LIN {X 0,Y 362.905,Z 706.892,A -85,B 0,C 180,E1 -22587.78,E2 -22587.78} C_VEL
LIN {X 0,Y 363.363,Z 707.01,A -85,B 0,C 180,E1 -22590,E2 -22590} C_VEL
LIN {X 0,Y 362.89,Z 706.909,A -85,B 0,C 180,E1 -22592.22,E2 -22592.22} C_VEL
LIN {X 0,Y 362.378,Z 706.638,A -85,B 0,C 180,E1 -22593.335,E2 -22593.335} C_VEL
LIN {X 0,Y 360.579,Z 706.015,A -85,B 0,C 180,E1 -22595.592,E2 -22595.592} C_VEL
LIN {X 0,Y 357.963,Z 704.809,A -85,B 0,C 180,E1 -22597.899,E2 -22597.899} C_VEL
LIN {X 0,Y 356.048,Z 703.774,A -85,B 0,C 180,E1 -22599.273,E2 -22599.273} C_VEL
LIN {X 0,Y 352.322,Z 701.531,A -85,B 0,C 180,E1 -22601.506,E2 -22601.506} C_VEL
LIN {X 0,Y 349.963,Z 699.883,A -85,B 0,C 180,E1 -22602.762,E2 -22602.762} C_VEL
LIN {X 0,Y 347.344,Z 697.848,A -85,B 0,C 180,E1 -22604.052,E2 -22604.052} C_VEL
LIN {X 0,Y 343.234,Z 695.3,A -85,B 0,C 180,E1 -22605.772,E2 -22605.772} C_VEL
LIN {X 0,Y 338.777,Z 692.643,A -85,B 0,C 180,E1 -22607.395,E2 -22607.395} C_VEL
LIN {X 0,Y 332.769,Z 688.318,A -85,B 0,C 180,E1 -22609.499,E2 -22609.499} C_VEL
LIN {X 0,Y 328.202,Z 685.08,A -85,B 0,C 180,E1 -22610.918,E2 -22610.918} C_VEL
LIN {X 0,Y 320.695,Z 679.914,A -85,B 0,C 180,E1 -22613.014,E2 -22613.014} C_VEL
LIN {X 0,Y 313.527,Z 674.664,A -85,B 0,C 180,E1 -22614.877,E2 -22614.877} C_VEL
LIN {X 0,Y 306.386,Z 669.423,A -85,B 0,C 180,E1 -22616.545,E2 -22616.545} C_VEL
LIN {X 0,Y 300.005,Z 664.622,A -85,B 0,C 180,E1 -22617.938,E2 -22617.938} C_VEL
LIN {X 0,Y 291.37,Z 657.885,A -85,B 0,C 180,E1 -22619.648,E2 -22619.648} C_VEL
LIN {X 0,Y 281.833,Z 650.578,A -85,B 0,C 180,E1 -22621.3,E2 -22621.3} C_VEL
LIN {X 0,Y 269.07,Z 639.844,A -85,B 0,C 180,E1 -22623.529,E2 -22623.529} C_VEL
LIN {X 0,Y 258.955,Z 630.539,A -85,B 0,C 180,E1 -22625.379,E2 -22625.379} C_VEL
LIN {X 0,Y 245.067,Z 616.202,A -85,B 0,C 180,E1 -22628.261,E2 -22628.261} C_VEL
LIN {X 0,Y 234.328,Z 603.001,A -85,B 0,C 180,E1 -22630.902,E2 -22630.902} C_VEL
LIN {X 0,Y 225.204,Z 588.908,A -85,B 0,C 180,E1 -22633.566,E2 -22633.566} C_VEL
LIN {X 0,Y 214.798,Z 569.008,A -85,B 0,C 180,E1 -22637.242,E2 -22637.242} C_VEL
LIN {X 0,Y 207.799,Z 557.073,A -85,B 0,C 180,E1 -22640.015,E2 -22640.015} C_VEL
LIN {X 0,Y 200.862,Z 546.571,A -85,B 0,C 180,E1 -22643.065,E2 -22643.065} C_VEL
LIN {X 0,Y 196.487,Z 540.686,A -85,B 0,C 180,E1 -22645.179,E2 -22645.179} C_VEL
LIN {X 0,Y 194.374,Z 537.758,A -85,B 0,C 180,E1 -22646.283,E2 -22646.283} C_VEL
LIN {X 0,Y 191.516,Z 533.827,A -85,B 0,C 180,E1 -22647.868,E2 -22647.868} C_VEL
LIN {X 0,Y 188.498,Z 530.398,A -85,B 0,C 180,E1 -22649.626,E2 -22649.626} C_VEL
LIN {X 0,Y 187.385,Z 528.546,A -85,B 0,C 180,E1 -22650.357,E2 -22650.357} C_VEL
LIN {X 0,Y 184.854,Z 526.226,A -85,B 0,C 180,E1 -22651.967,E2 -22651.967} C_VEL
LIN {X 0,Y 183.022,Z 523.18,A -85,B 0,C 180,E1 -22653.335,E2 -22653.335} C_VEL
LIN {X 0,Y 180.33,Z 521.243,A -85,B 0,C 180,E1 -22655.289,E2 -22655.289} C_VEL
LIN {X 0,Y 178.835,Z 518.728,A -85,B 0,C 180,E1 -22656.65,E2 -22656.65} C_VEL
LIN {X 0,Y 178.593,Z 517.589,A -85,B 0,C 180,E1 -22657.516,E2 -22657.516} C_VEL
LIN {X 0,Y 178.645,Z 517.32,A -85,B 0,C 180,E1 -22661.657,E2 -22661.657} C_VEL
LIN {X 0,Y 178.652,Z 517.357,A -85,B 0,C 180,E1 -22666.349,E2 -22666.349} C_VEL
LIN {X 0,Y 178.907,Z 517.281,A -85,B 0,C 180,E1 -22670.961,E2 -22670.961} C_VEL
LIN {X 0,Y 178.862,Z 517.301,A -85,B 0,C 180,E1 -22675.494,E2 -22675.494} C_VEL
LIN {X 0,Y 179.366,Z 517.233,A -85,B 0,C 180,E1 -22680.001,E2 -22680.001} C_VEL
LIN {X 0,Y 178.866,Z 517.288,A -85,B 0,C 180,E1 -22684.508,E2 -22684.508} C_VEL
LIN {X 0,Y 178.956,Z 517.309,A -85,B 0,C 180,E1 -22689.039,E2 -22689.039} C_VEL
LIN {X 0,Y 178.657,Z 517.313,A -85,B 0,C 180,E1 -22693.653,E2 -22693.653} C_VEL
LIN {X 0,Y 178.619,Z 517.329,A -85,B 0,C 180,E1 -22699.215,E2 -22699.215} C_VEL
LIN {X 0,Y 178.603,Z 517.694,A -85,B 0,C 180,E1 -22702.257,E2 -22702.257} C_VEL
LIN {X 0,Y 178.855,Z 518.824,A -85,B 0,C 180,E1 -22702.986,E2 -22702.986} C_VEL
LIN {X 0,Y 180.307,Z 521.22,A -85,B 0,C 180,E1 -22704.3,E2 -22704.3} C_VEL
LIN {X 0,Y 182.575,Z 522.942,A -85,B 0,C 180,E1 -22705.969,E2 -22705.969} C_VEL
LIN {X 0,Y 183.29,Z 523.542,A -85,B 0,C 180,E1 -22706.472,E2 -22706.472} C_VEL
LIN {X 0,Y 185.238,Z 526.708,A -85,B 0,C 180,E1 -22707.904,E2 -22707.904} C_VEL
LIN {X 0,Y 187.677,Z 528.97,A -85,B 0,C 180,E1 -22709.44,E2 -22709.44} C_VEL
LIN {X 0,Y 190.188,Z 532.55,A -85,B 0,C 180,E1 -22711.001,E2 -22711.001} C_VEL
LIN {X 0,Y 191.704,Z 534.216,A -85,B 0,C 180,E1 -22711.856,E2 -22711.856} C_VEL
LIN {X 0,Y 194.572,Z 537.949,A -85,B 0,C 180,E1 -22713.425,E2 -22713.425} C_VEL
LIN {X 0,Y 198.501,Z 544.029,A -85,B 0,C 180,E1 -22715.465,E2 -22715.465} C_VEL
LIN {X 0,Y 203.758,Z 553.106,A -85,B 0,C 180,E1 -22717.987,E2 -22717.987} C_VEL
LIN {X 0,Y 209.85,Z 564.904,A -85,B 0,C 180,E1 -22720.663,E2 -22720.663} C_VEL
LIN {X 0,Y 215.674,Z 577.872,A -85,B 0,C 180,E1 -22723.042,E2 -22723.042} C_VEL
LIN {X 0,Y 220.269,Z 589.701,A -85,B 0,C 180,E1 -22724.835,E2 -22724.835} C_VEL
LIN {X 0,Y 216.464,Z 650.604,A -85,B 0,C 180,E1 -22726.656,E2 -22726.656} C_VEL
LIN {X 0,Y 215.159,Z 662.058,A -85,B 0,C 180,E1 -22727.171,E2 -22727.171} C_VEL
LIN {X 0,Y 213.613,Z 671.685,A -85,B 0,C 180,E1 -22727.748,E2 -22727.748} C_VEL
LIN {X 0,Y 211.279,Z 682.832,A -85,B 0,C 180,E1 -22728.616,E2 -22728.616} C_VEL
LIN {X 0,Y 208.839,Z 692.8,A -85,B 0,C 180,E1 -22729.624,E2 -22729.624} C_VEL
LIN {X 0,Y 206.009,Z 702.716,A -85,B 0,C 180,E1 -22730.868,E2 -22730.868} C_VEL
LIN {X 0,Y 202.81,Z 712.435,A -85,B 0,C 180,E1 -22732.356,E2 -22732.356} C_VEL
LIN {X 0,Y 199.59,Z 721.567,A -85,B 0,C 180,E1 -22734.086,E2 -22734.086} C_VEL
LIN {X 0,Y 195.973,Z 730.873,A -85,B 0,C 180,E1 -22736.231,E2 -22736.231} C_VEL
LIN {X 0,Y 192.94,Z 737.844,A -85,B 0,C 180,E1 -22738.119,E2 -22738.119} C_VEL
LIN {X 0,Y 189.528,Z 745.364,A -85,B 0,C 180,E1 -22740.573,E2 -22740.573} C_VEL
LIN {X 0,Y 185.961,Z 752.975,A -85,B 0,C 180,E1 -22743.637,E2 -22743.637} C_VEL
LIN {X 0,Y 183.399,Z 758.378,A -85,B 0,C 180,E1 -22746.274,E2 -22746.274} C_VEL
LIN {X 0,Y 180.937,Z 763.817,A -85,B 0,C 180,E1 -22749.539,E2 -22749.539} C_VEL
LIN {X 0,Y 178.939,Z 768.266,A -85,B 0,C 180,E1 -22752.869,E2 -22752.869} C_VEL
LIN {X 0,Y 178.633,Z 768.942,A -85,B 0,C 180,E1 -22753.466,E2 -22753.466} C_VEL
LIN {X 0,Y 177.192,Z 770.925,A -85,B 0,C 180,E1 -22755.207,E2 -22755.207} C_VEL
LIN {X 0,Y 173.38,Z 773.511,A -85,B 0,C 180,E1 -22758.07,E2 -22758.07} C_VEL
LIN {X 0,Y 170.438,Z 775.159,A -85,B 0,C 180,E1 -22760.475,E2 -22760.475} C_VEL
LIN {X 0,Y 169.124,Z 776.109,A -85,B 0,C 180,E1 -22762.401,E2 -22762.401} C_VEL
LIN {X 0,Y 168.971,Z 776.341,A -85,B 0,C 180,E1 -22763.064,E2 -22763.064} C_VEL
LIN {X 0,Y 168.89,Z 777.565,A -85,B 0,C 180,E1 -22767.615,E2 -22767.615} C_VEL
LIN {X 0,Y 168.989,Z 777.822,A -85,B 0,C 180,E1 -22770,E2 -22770} C_VEL
LIN {X 0,Y 168.876,Z 777.085,A -85,B 0,C 180,E1 -22774.774,E2 -22774.774} C_VEL
LIN {X 0,Y 168.995,Z 776.261,A -85,B 0,C 180,E1 -22777.167,E2 -22777.167} C_VEL
LIN {X 0,Y 169.781,Z 773.563,A -85,B 0,C 180,E1 -22781.945,E2 -22781.945} C_VEL
LIN {X 0,Y 171.508,Z 769.334,A -85,B 0,C 180,E1 -22786.669,E2 -22786.669} C_VEL
LIN {X 0,Y 173.456,Z 765.197,A -85,B 0,C 180,E1 -22790.145,E2 -22790.145} C_VEL
LIN {X 0,Y 175.898,Z 760.093,A -85,B 0,C 180,E1 -22793.549,E2 -22793.549} C_VEL
LIN {X 0,Y 178.995,Z 753.913,A -85,B 0,C 180,E1 -22796.841,E2 -22796.841} C_VEL
LIN {X 0,Y 182.03,Z 747.84,A -85,B 0,C 180,E1 -22799.489,E2 -22799.489} C_VEL
LIN {X 0,Y 185.435,Z 740.767,A -85,B 0,C 180,E1 -22802.045,E2 -22802.045} C_VEL
LIN {X 0,Y 188.506,Z 734.31,A -85,B 0,C 180,E1 -22804.002,E2 -22804.002} C_VEL
LIN {X 0,Y 192.369,Z 725.334,A -85,B 0,C 180,E1 -22806.264,E2 -22806.264} C_VEL
LIN {X 0,Y 195.922,Z 715.957,A -85,B 0,C 180,E1 -22808.226,E2 -22808.226} C_VEL
LIN {X 0,Y 199.134,Z 706.91,A -85,B 0,C 180,E1 -22809.767,E2 -22809.767} C_VEL
LIN {X 0,Y 202.473,Z 696.107,A -85,B 0,C 180,E1 -22811.261,E2 -22811.261} C_VEL
LIN {X 0,Y 205.254,Z 685.854,A -85,B 0,C 180,E1 -22812.384,E2 -22812.384} C_VEL
LIN {X 0,Y 207.849,Z 674.205,A -85,B 0,C 180,E1 -22813.378,E2 -22813.378} C_VEL
LIN {X 0,Y 209.834,Z 662.77,A -85,B 0,C 180,E1 -22814.108,E2 -22814.108} C_VEL
LIN {X 0,Y 211.198,Z 651.913,A -85,B 0,C 180,E1 -22814.603,E2 -22814.603} C_VEL
LIN {X 0,Y 212.886,Z 628.702,A -85,B 0,C 180,E1 -22815.328,E2 -22815.328} C_VEL
LIN {X 0,Y 215.147,Z 591.855,A -85,B 0,C 180,E1 -22816.442,E2 -22816.442} C_VEL
LIN {X 0,Y 210.265,Z 579.231,A -85,B 0,C 180,E1 -22818.481,E2 -22818.481} C_VEL
LIN {X 0,Y 204.814,Z 567.17,A -85,B 0,C 180,E1 -22820.871,E2 -22820.871} C_VEL
LIN {X 0,Y 199.071,Z 556.016,A -85,B 0,C 180,E1 -22823.59,E2 -22823.59} C_VEL
LIN {X 0,Y 193.918,Z 547.035,A -85,B 0,C 180,E1 -22826.272,E2 -22826.272} C_VEL
LIN {X 0,Y 191.631,Z 543.666,A -85,B 0,C 180,E1 -22827.531,E2 -22827.531} C_VEL
LIN {X 0,Y 188.143,Z 539.098,A -85,B 0,C 180,E1 -22829.56,E2 -22829.56} C_VEL
LIN {X 0,Y 185.338,Z 535.278,A -85,B 0,C 180,E1 -22831.356,E2 -22831.356} C_VEL
LIN {X 0,Y 182.1,Z 531.683,A -85,B 0,C 180,E1 -22833.573,E2 -22833.573} C_VEL
LIN {X 0,Y 180.96,Z 529.723,A -85,B 0,C 180,E1 -22834.477,E2 -22834.477} C_VEL
LIN {X 0,Y 178.143,Z 527.388,A -85,B 0,C 180,E1 -22836.658,E2 -22836.658} C_VEL
LIN {X 0,Y 176.353,Z 524.222,A -85,B 0,C 180,E1 -22838.368,E2 -22838.368} C_VEL
LIN {X 0,Y 173.51,Z 522.23,A -85,B 0,C 180,E1 -22841.092,E2 -22841.092} C_VEL
LIN {X 0,Y 171.922,Z 519.752,A -85,B 0,C 180,E1 -22843.065,E2 -22843.065} C_VEL
LIN {X 0,Y 171.653,Z 518.682,A -85,B 0,C 180,E1 -22843.955,E2 -22843.955} C_VEL
LIN {X 0,Y 171.579,Z 518.242,A -85,B 0,C 180,E1 -22845.772,E2 -22845.772} C_VEL
LIN {X 0,Y 171.885,Z 518.196,A -85,B 0,C 180,E1 -22850.586,E2 -22850.586} C_VEL
LIN {X 0,Y 171.815,Z 518.164,A -85,B 0,C 180,E1 -22855.306,E2 -22855.306} C_VEL
LIN {X 0,Y 172.328,Z 518.108,A -85,B 0,C 180,E1 -22859.999,E2 -22859.999} C_VEL
LIN {X 0,Y 171.809,Z 518.181,A -85,B 0,C 180,E1 -22864.692,E2 -22864.692} C_VEL
LIN {X 0,Y 171.844,Z 518.159,A -85,B 0,C 180,E1 -22869.414,E2 -22869.414} C_VEL
LIN {X 0,Y 171.607,Z 518.454,A -85,B 0,C 180,E1 -22876.047,E2 -22876.047} C_VEL
LIN {X 0,Y 171.876,Z 519.587,A -85,B 0,C 180,E1 -22877.243,E2 -22877.243} C_VEL
LIN {X 0,Y 173.784,Z 522.574,A -85,B 0,C 180,E1 -22879.602,E2 -22879.602} C_VEL
LIN {X 0,Y 176.557,Z 524.493,A -85,B 0,C 180,E1 -22882.218,E2 -22882.218} C_VEL
LIN {X 0,Y 178.285,Z 527.504,A -85,B 0,C 180,E1 -22883.85,E2 -22883.85} C_VEL
LIN {X 0,Y 180.95,Z 529.712,A -85,B 0,C 180,E1 -22885.908,E2 -22885.908} C_VEL
LIN {X 0,Y 183.514,Z 533.532,A -85,B 0,C 180,E1 -22887.84,E2 -22887.84} C_VEL
LIN {X 0,Y 185.378,Z 535.313,A -85,B 0,C 180,E1 -22889.061,E2 -22889.061} C_VEL
LIN {X 0,Y 187.977,Z 538.94,A -85,B 0,C 180,E1 -22890.735,E2 -22890.735} C_VEL
LIN {X 0,Y 189.369,Z 540.617,A -85,B 0,C 180,E1 -22891.562,E2 -22891.562} C_VEL
LIN {X 0,Y 193.048,Z 545.647,A -85,B 0,C 180,E1 -22893.644,E2 -22893.644} C_VEL
LIN {X 0,Y 198.254,Z 552.943,A -85,B 0,C 180,E1 -22896.299,E2 -22896.299} C_VEL
LIN {X 0,Y 205.149,Z 563.699,A -85,B 0,C 180,E1 -22899.448,E2 -22899.448} C_VEL
LIN {X 0,Y 212.19,Z 576.289,A -85,B 0,C 180,E1 -22902.346,E2 -22902.346} C_VEL
LIN {X 0,Y 222.747,Z 596.607,A -85,B 0,C 180,E1 -22906.165,E2 -22906.165} C_VEL
LIN {X 0,Y 231.199,Z 609.336,A -85,B 0,C 180,E1 -22908.676,E2 -22908.676} C_VEL
LIN {X 0,Y 242.228,Z 622.966,A -85,B 0,C 180,E1 -22911.456,E2 -22911.456} C_VEL
LIN {X 0,Y 259.155,Z 640.207,A -85,B 0,C 180,E1 -22915.013,E2 -22915.013} C_VEL
LIN {X 0,Y 272.396,Z 651.933,A -85,B 0,C 180,E1 -22917.55,E2 -22917.55} C_VEL
LIN {X 0,Y 284.672,Z 661.727,A -85,B 0,C 180,E1 -22919.776,E2 -22919.776} C_VEL
LIN {X 0,Y 292.731,Z 667.984,A -85,B 0,C 180,E1 -22921.304,E2 -22921.304} C_VEL
LIN {X 0,Y 300.156,Z 673.487,A -85,B 0,C 180,E1 -22922.84,E2 -22922.84} C_VEL
LIN {X 0,Y 308.356,Z 679.696,A -85,B 0,C 180,E1 -22924.746,E2 -22924.746} C_VEL
LIN {X 0,Y 314.653,Z 684.211,A -85,B 0,C 180,E1 -22926.313,E2 -22926.313} C_VEL
LIN {X 0,Y 321.531,Z 689.206,A -85,B 0,C 180,E1 -22928.187,E2 -22928.187} C_VEL
LIN {X 0,Y 327.367,Z 693.076,A -85,B 0,C 180,E1 -22929.911,E2 -22929.911} C_VEL
LIN {X 0,Y 332.932,Z 697.209,A -85,B 0,C 180,E1 -22931.789,E2 -22931.789} C_VEL
LIN {X 0,Y 337.364,Z 700.135,A -85,B 0,C 180,E1 -22933.388,E2 -22933.388} C_VEL
LIN {X 0,Y 341.829,Z 702.742,A -85,B 0,C 180,E1 -22935.085,E2 -22935.085} C_VEL
LIN {X 0,Y 346.118,Z 705.829,A -85,B 0,C 180,E1 -22937.094,E2 -22937.094} C_VEL
LIN {X 0,Y 350.333,Z 708.69,A -85,B 0,C 180,E1 -22939.411,E2 -22939.411} C_VEL
LIN {X 0,Y 352.63,Z 710.005,A -85,B 0,C 180,E1 -22940.826,E2 -22940.826} C_VEL
LIN {X 0,Y 354.633,Z 711.024,A -85,B 0,C 180,E1 -22942.252,E2 -22942.252} C_VEL
LIN {X 0,Y 357.009,Z 712.133,A -85,B 0,C 180,E1 -22944.351,E2 -22944.351} C_VEL
LIN {X 0,Y 358.829,Z 712.796,A -85,B 0,C 180,E1 -22946.632,E2 -22946.632} C_VEL
LIN {X 0,Y 359.67,Z 713.222,A -85,B 0,C 180,E1 -22948.88,E2 -22948.88} C_VEL
LIN {X 0,Y 359.842,Z 713.165,A -85,B 0,C 180,E1 -22950,E2 -22950} C_VEL
LIN {X 0,Y 359.359,Z 713.05,A -85,B 0,C 180,E1 -22952.242,E2 -22952.242} C_VEL
LIN {X 0,Y 358.825,Z 712.794,A -85,B 0,C 180,E1 -22953.368,E2 -22953.368} C_VEL
LIN {X 0,Y 356.992,Z 712.124,A -85,B 0,C 180,E1 -22955.649,E2 -22955.649} C_VEL
LIN {X 0,Y 354.314,Z 710.883,A -85,B 0,C 180,E1 -22957.981,E2 -22957.981} C_VEL
LIN {X 0,Y 352.642,Z 709.991,A -85,B 0,C 180,E1 -22959.174,E2 -22959.174} C_VEL
LIN {X 0,Y 350.346,Z 708.631,A -85,B 0,C 180,E1 -22960.6,E2 -22960.6} C_VEL
LIN {X 0,Y 346.092,Z 705.787,A -85,B 0,C 180,E1 -22962.913,E2 -22962.913} C_VEL
LIN {X 0,Y 343.467,Z 703.775,A -85,B 0,C 180,E1 -22964.214,E2 -22964.214} C_VEL
LIN {X 0,Y 340.187,Z 701.714,A -85,B 0,C 180,E1 -22965.579,E2 -22965.579} C_VEL
LIN {X 0,Y 334.605,Z 698.353,A -85,B 0,C 180,E1 -22967.619,E2 -22967.619} C_VEL
LIN {X 0,Y 330.333,Z 695.362,A -85,B 0,C 180,E1 -22969.093,E2 -22969.093} C_VEL
LIN {X 0,Y 325.682,Z 691.857,A -85,B 0,C 180,E1 -22970.609,E2 -22970.609} C_VEL
LIN {X 0,Y 319.311,Z 687.685,A -85,B 0,C 180,E1 -22972.422,E2 -22972.422} C_VEL
LIN {X 0,Y 311.929,Z 682.108,A -85,B 0,C 180,E1 -22974.4,E2 -22974.4} C_VEL
LIN {X 0,Y 305.046,Z 677.258,A -85,B 0,C 180,E1 -22976.037,E2 -22976.037} C_VEL
LIN {X 0,Y 297.201,Z 671.321,A -85,B 0,C 180,E1 -22977.783,E2 -22977.783} C_VEL
LIN {X 0,Y 289.955,Z 665.849,A -85,B 0,C 180,E1 -22979.242,E2 -22979.242} C_VEL
LIN {X 0,Y 277.47,Z 656.096,A -85,B 0,C 180,E1 -22981.52,E2 -22981.52} C_VEL
LIN {X 0,Y 265.317,Z 645.767,A -85,B 0,C 180,E1 -22983.797,E2 -22983.797} C_VEL
LIN {X 0,Y 255.079,Z 636.167,A -85,B 0,C 180,E1 -22985.808,E2 -22985.808} C_VEL
LIN {X 0,Y 241.373,Z 621.944,A -85,B 0,C 180,E1 -22988.745,E2 -22988.745} C_VEL
LIN {X 0,Y 230.564,Z 608.539,A -85,B 0,C 180,E1 -22991.496,E2 -22991.496} C_VEL
LIN {X 0,Y 221.184,Z 593.901,A -85,B 0,C 180,E1 -22994.348,E2 -22994.348} C_VEL
LIN {X 0,Y 210.835,Z 573.743,A -85,B 0,C 180,E1 -22998.19,E2 -22998.19} C_VEL
LIN {X 0,Y 204.299,Z 562.343,A -85,B 0,C 180,E1 -23000.919,E2 -23000.919} C_VEL
LIN {X 0,Y 197.628,Z 552.023,A -85,B 0,C 180,E1 -23004.007,E2 -23004.007} C_VEL
LIN {X 0,Y 191.86,Z 543.943,A -85,B 0,C 180,E1 -23007.013,E2 -23007.013} C_VEL
LIN {X 0,Y 188.365,Z 539.328,A -85,B 0,C 180,E1 -23009.037,E2 -23009.037} C_VEL
LIN {X 0,Y 185.644,Z 535.802,A -85,B 0,C 180,E1 -23010.752,E2 -23010.752} C_VEL
LIN {X 0,Y 184.812,Z 534.712,A -85,B 0,C 180,E1 -23011.307,E2 -23011.307} C_VEL
LIN {X 0,Y 182.196,Z 531.838,A -85,B 0,C 180,E1 -23013.107,E2 -23013.107} C_VEL
LIN {X 0,Y 180.95,Z 529.712,A -85,B 0,C 180,E1 -23014.092,E2 -23014.092} C_VEL
LIN {X 0,Y 178.284,Z 527.506,A -85,B 0,C 180,E1 -23016.149,E2 -23016.149} C_VEL
LIN {X 0,Y 176.557,Z 524.495,A -85,B 0,C 180,E1 -23017.782,E2 -23017.782} C_VEL
LIN {X 0,Y 173.306,Z 522.031,A -85,B 0,C 180,E1 -23020.92,E2 -23020.92} C_VEL
LIN {X 0,Y 171.673,Z 518.848,A -85,B 0,C 180,E1 -23023.349,E2 -23023.349} C_VEL
LIN {X 0,Y 171.555,Z 518.256,A -85,B 0,C 180,E1 -23025.166,E2 -23025.166} C_VEL
LIN {X 0,Y 171.844,Z 518.159,A -85,B 0,C 180,E1 -23030.586,E2 -23030.586} C_VEL
LIN {X 0,Y 171.811,Z 518.181,A -85,B 0,C 180,E1 -23035.308,E2 -23035.308} C_VEL
LIN {X 0,Y 172.328,Z 518.108,A -85,B 0,C 180,E1 -23040.001,E2 -23040.001} C_VEL
LIN {X 0,Y 171.815,Z 518.164,A -85,B 0,C 180,E1 -23044.694,E2 -23044.694} C_VEL
LIN {X 0,Y 171.885,Z 518.196,A -85,B 0,C 180,E1 -23049.414,E2 -23049.414} C_VEL
LIN {X 0,Y 171.588,Z 518.384,A -85,B 0,C 180,E1 -23055.441,E2 -23055.441} C_VEL
LIN {X 0,Y 171.806,Z 519.369,A -85,B 0,C 180,E1 -23056.717,E2 -23056.717} C_VEL
LIN {X 0,Y 173.255,Z 521.963,A -85,B 0,C 180,E1 -23058.63,E2 -23058.63} C_VEL
LIN {X 0,Y 175.743,Z 523.912,A -85,B 0,C 180,E1 -23061.096,E2 -23061.096} C_VEL
LIN {X 0,Y 176.568,Z 524.494,A -85,B 0,C 180,E1 -23061.835,E2 -23061.835} C_VEL
LIN {X 0,Y 178.143,Z 527.388,A -85,B 0,C 180,E1 -23063.342,E2 -23063.342} C_VEL
LIN {X 0,Y 181.266,Z 530.204,A -85,B 0,C 180,E1 -23065.765,E2 -23065.765} C_VEL
LIN {X 0,Y 183.689,Z 533.679,A -85,B 0,C 180,E1 -23067.564,E2 -23067.564} C_VEL
LIN {X 0,Y 185.421,Z 535.389,A -85,B 0,C 180,E1 -23068.699,E2 -23068.699} C_VEL
LIN {X 0,Y 188.143,Z 539.098,A -85,B 0,C 180,E1 -23070.44,E2 -23070.44} C_VEL
LIN {X 0,Y 189.535,Z 540.938,A -85,B 0,C 180,E1 -23071.274,E2 -23071.274} C_VEL
LIN {X 0,Y 193.055,Z 545.642,A -85,B 0,C 180,E1 -23073.254,E2 -23073.254} C_VEL
LIN {X 0,Y 197.657,Z 553.388,A -85,B 0,C 180,E1 -23075.695,E2 -23075.695} C_VEL
LIN {X 0,Y 204.062,Z 565.602,A -85,B 0,C 180,E1 -23078.785,E2 -23078.785} C_VEL
LIN {X 0,Y 209.42,Z 577.282,A -85,B 0,C 180,E1 -23081.16,E2 -23081.16} C_VEL
LIN {X 0,Y 214.142,Z 589.072,A -85,B 0,C 180,E1 -23083.143,E2 -23083.143} C_VEL
LIN {X 0,Y 215.156,Z 591.847,A -85,B 0,C 180,E1 -23083.56,E2 -23083.56} C_VEL
LIN {X 0,Y 211.303,Z 650.989,A -85,B 0,C 180,E1 -23085.358,E2 -23085.358} C_VEL
LIN {X 0,Y 209.851,Z 662.771,A -85,B 0,C 180,E1 -23085.896,E2 -23085.896} C_VEL
LIN {X 0,Y 208.161,Z 672.847,A -85,B 0,C 180,E1 -23086.537,E2 -23086.537} C_VEL
LIN {X 0,Y 206.015,Z 682.635,A -85,B 0,C 180,E1 -23087.312,E2 -23087.312} C_VEL
LIN {X 0,Y 203.467,Z 692.601,A -85,B 0,C 180,E1 -23088.325,E2 -23088.325} C_VEL
LIN {X 0,Y 200.538,Z 702.517,A -85,B 0,C 180,E1 -23089.584,E2 -23089.584} C_VEL
LIN {X 0,Y 197.22,Z 712.236,A -85,B 0,C 180,E1 -23091.093,E2 -23091.093} C_VEL
LIN {X 0,Y 194.273,Z 720.289,A -85,B 0,C 180,E1 -23092.61,E2 -23092.61} C_VEL
LIN {X 0,Y 190.853,Z 728.855,A -85,B 0,C 180,E1 -23094.552,E2 -23094.552} C_VEL
LIN {X 0,Y 186.923,Z 737.645,A -85,B 0,C 180,E1 -23096.964,E2 -23096.964} C_VEL
LIN {X 0,Y 183.334,Z 745.164,A -85,B 0,C 180,E1 -23099.475,E2 -23099.475} C_VEL
LIN {X 0,Y 179.59,Z 752.776,A -85,B 0,C 180,E1 -23102.625,E2 -23102.625} C_VEL
LIN {X 0,Y 176.872,Z 758.179,A -85,B 0,C 180,E1 -23105.342,E2 -23105.342} C_VEL
LIN {X 0,Y 174.227,Z 763.616,A -85,B 0,C 180,E1 -23108.713,E2 -23108.713} C_VEL
LIN {X 0,Y 172.115,Z 768.066,A -85,B 0,C 180,E1 -23112.167,E2 -23112.167} C_VEL
LIN {X 0,Y 170.472,Z 771.615,A -85,B 0,C 180,E1 -23115.679,E2 -23115.679} C_VEL
LIN {X 0,Y 169.781,Z 773.563,A -85,B 0,C 180,E1 -23118.055,E2 -23118.055} C_VEL
LIN {X 0,Y 168.971,Z 776.341,A -85,B 0,C 180,E1 -23123.064,E2 -23123.064} C_VEL
LIN {X 0,Y 168.165,Z 777.042,A -85,B 0,C 180,E1 -23125.045,E2 -23125.045} C_VEL
LIN {X 0,Y 166.531,Z 777.44,A -85,B 0,C 180,E1 -23127.001,E2 -23127.001} C_VEL
LIN {X 0,Y 162.848,Z 777.561,A -85,B 0,C 180,E1 -23130.986,E2 -23130.986} C_VEL
LIN {X 0,Y 161.837,Z 777.303,A -85,B 0,C 180,E1 -23133.073,E2 -23133.073} C_VEL
LIN {X 0,Y 161.758,Z 777.119,A -85,B 0,C 180,E1 -23133.78,E2 -23133.78} C_VEL
LIN {X 0,Y 161.931,Z 776.062,A -85,B 0,C 180,E1 -23137.481,E2 -23137.481} C_VEL
LIN {X 0,Y 162.791,Z 773.363,A -85,B 0,C 180,E1 -23142.466,E2 -23142.466} C_VEL
LIN {X 0,Y 164.669,Z 769.135,A -85,B 0,C 180,E1 -23147.382,E2 -23147.382} C_VEL
LIN {X 0,Y 166.759,Z 764.997,A -85,B 0,C 180,E1 -23150.991,E2 -23150.991} C_VEL
LIN {X 0,Y 168.599,Z 761.368,A -85,B 0,C 180,E1 -23153.626,E2 -23153.626} C_VEL
LIN {X 0,Y 172.058,Z 754.852,A -85,B 0,C 180,E1 -23157.356,E2 -23157.356} C_VEL
LIN {X 0,Y 175.847,Z 747.64,A -85,B 0,C 180,E1 -23160.635,E2 -23160.635} C_VEL
LIN {X 0,Y 179.445,Z 740.568,A -85,B 0,C 180,E1 -23163.251,E2 -23163.251} C_VEL
LIN {X 0,Y 182.638,Z 734.112,A -85,B 0,C 180,E1 -23165.253,E2 -23165.253} C_VEL
LIN {X 0,Y 186.99,Z 724.34,A -85,B 0,C 180,E1 -23167.738,E2 -23167.738} C_VEL
LIN {X 0,Y 190.371,Z 715.759,A -85,B 0,C 180,E1 -23169.554,E2 -23169.554} C_VEL
LIN {X 0,Y 193.725,Z 706.711,A -85,B 0,C 180,E1 -23171.112,E2 -23171.112} C_VEL
LIN {X 0,Y 197.187,Z 695.909,A -85,B 0,C 180,E1 -23172.623,E2 -23172.623} C_VEL
LIN {X 0,Y 200.064,Z 685.656,A -85,B 0,C 180,E1 -23173.755,E2 -23173.755} C_VEL
LIN {X 0,Y 202.736,Z 674.007,A -85,B 0,C 180,E1 -23174.759,E2 -23174.759} C_VEL
LIN {X 0,Y 204.8,Z 662.572,A -85,B 0,C 180,E1 -23175.489,E2 -23175.489} C_VEL
LIN {X 0,Y 206.269,Z 651.209,A -85,B 0,C 180,E1 -23176.002,E2 -23176.002} C_VEL
LIN {X 0,Y 208.217,Z 624.261,A -85,B 0,C 180,E1 -23176.852,E2 -23176.852} C_VEL
LIN {X 0,Y 210.149,Z 594.036,A -85,B 0,C 180,E1 -23177.776,E2 -23177.776} C_VEL
LIN {X 0,Y 205.579,Z 582.156,A -85,B 0,C 180,E1 -23179.813,E2 -23179.813} C_VEL
LIN {X 0,Y 200.168,Z 569.984,A -85,B 0,C 180,E1 -23182.362,E2 -23182.362} C_VEL
LIN {X 0,Y 194.218,Z 558.324,A -85,B 0,C 180,E1 -23185.416,E2 -23185.416} C_VEL
LIN {X 0,Y 189.519,Z 550.238,A -85,B 0,C 180,E1 -23188.078,E2 -23188.078} C_VEL
LIN {X 0,Y 185.524,Z 545.038,A -85,B 0,C 180,E1 -23190.496,E2 -23190.496} C_VEL
LIN {X 0,Y 182.586,Z 540.985,A -85,B 0,C 180,E1 -23192.489,E2 -23192.489} C_VEL
LIN {X 0,Y 179.793,Z 537.674,A -85,B 0,C 180,E1 -23194.532,E2 -23194.532} C_VEL
LIN {X 0,Y 178.764,Z 536.145,A -85,B 0,C 180,E1 -23195.371,E2 -23195.371} C_VEL
LIN {X 0,Y 175.971,Z 533.397,A -85,B 0,C 180,E1 -23197.701,E2 -23197.701} C_VEL
LIN {X 0,Y 174.641,Z 530.914,A -85,B 0,C 180,E1 -23199.055,E2 -23199.055} C_VEL
LIN {X 0,Y 171.899,Z 528.794,A -85,B 0,C 180,E1 -23201.835,E2 -23201.835} C_VEL
LIN {X 0,Y 170.209,Z 525.988,A -85,B 0,C 180,E1 -23204.046,E2 -23204.046} C_VEL
LIN {X 0,Y 169.754,Z 525.275,A -85,B 0,C 180,E1 -23204.695,E2 -23204.695} C_VEL
LIN {X 0,Y 166.555,Z 522.95,A -85,B 0,C 180,E1 -23209.885,E2 -23209.885} C_VEL
LIN {X 0,Y 164.948,Z 519.938,A -85,B 0,C 180,E1 -23215.417,E2 -23215.417} C_VEL
LIN {X 0,Y 165.162,Z 519.192,A -85,B 0,C 180,E1 -23218.78,E2 -23218.78} C_VEL
LIN {X 0,Y 165.291,Z 519.107,A -85,B 0,C 180,E1 -23219.999,E2 -23219.999} C_VEL
LIN {X 0,Y 164.923,Z 519.729,A -85,B 0,C 180,E1 -23224.276,E2 -23224.276} C_VEL
LIN {X 0,Y 165.647,Z 521.678,A -85,B 0,C 180,E1 -23228.231,E2 -23228.231} C_VEL
LIN {X 0,Y 168.443,Z 524.604,A -85,B 0,C 180,E1 -23233.88,E2 -23233.88} C_VEL
LIN {X 0,Y 170.016,Z 525.504,A -85,B 0,C 180,E1 -23236.047,E2 -23236.047} C_VEL
LIN {X 0,Y 171.829,Z 528.735,A -85,B 0,C 180,E1 -23238.479,E2 -23238.479} C_VEL
LIN {X 0,Y 174.26,Z 530.741,A -85,B 0,C 180,E1 -23240.991,E2 -23240.991} C_VEL
LIN {X 0,Y 174.877,Z 531.394,A -85,B 0,C 180,E1 -23241.589,E2 -23241.589} C_VEL
LIN {X 0,Y 177,Z 534.637,A -85,B 0,C 180,E1 -23243.607,E2 -23243.607} C_VEL
LIN {X 0,Y 179.317,Z 536.813,A -85,B 0,C 180,E1 -23245.462,E2 -23245.462} C_VEL
LIN {X 0,Y 181.917,Z 540.386,A -85,B 0,C 180,E1 -23247.448,E2 -23247.448} C_VEL
LIN {X 0,Y 183.249,Z 541.902,A -85,B 0,C 180,E1 -23248.37,E2 -23248.37} C_VEL
LIN {X 0,Y 186.209,Z 545.756,A -85,B 0,C 180,E1 -23250.317,E2 -23250.317} C_VEL
LIN {X 0,Y 192.676,Z 554.811,A -85,B 0,C 180,E1 -23254.08,E2 -23254.08} C_VEL
LIN {X 0,Y 199.017,Z 564.587,A -85,B 0,C 180,E1 -23257.287,E2 -23257.287} C_VEL
LIN {X 0,Y 204.885,Z 574.66,A -85,B 0,C 180,E1 -23259.95,E2 -23259.95} C_VEL
LIN {X 0,Y 210.616,Z 585.803,A -85,B 0,C 180,E1 -23262.347,E2 -23262.347} C_VEL
LIN {X 0,Y 218.557,Z 601.311,A -85,B 0,C 180,E1 -23265.307,E2 -23265.307} C_VEL
LIN {X 0,Y 227.215,Z 614.565,A -85,B 0,C 180,E1 -23267.999,E2 -23267.999} C_VEL
LIN {X 0,Y 238.202,Z 628.281,A -85,B 0,C 180,E1 -23270.878,E2 -23270.878} C_VEL
LIN {X 0,Y 252.675,Z 643.349,A -85,B 0,C 180,E1 -23274.104,E2 -23274.104} C_VEL
LIN {X 0,Y 266.116,Z 655.832,A -85,B 0,C 180,E1 -23276.924,E2 -23276.924} C_VEL
LIN {X 0,Y 280.639,Z 667.57,A -85,B 0,C 180,E1 -23279.766,E2 -23279.766} C_VEL
LIN {X 0,Y 289.747,Z 674.632,A -85,B 0,C 180,E1 -23281.53,E2 -23281.53} C_VEL
LIN {X 0,Y 296.148,Z 679.365,A -85,B 0,C 180,E1 -23282.862,E2 -23282.862} C_VEL
LIN {X 0,Y 303.536,Z 684.937,A -85,B 0,C 180,E1 -23284.553,E2 -23284.553} C_VEL
LIN {X 0,Y 311.281,Z 690.531,A -85,B 0,C 180,E1 -23286.472,E2 -23286.472} C_VEL
LIN {X 0,Y 317.758,Z 695.206,A -85,B 0,C 180,E1 -23288.267,E2 -23288.267} C_VEL
LIN {X 0,Y 324.174,Z 699.542,A -85,B 0,C 180,E1 -23290.175,E2 -23290.175} C_VEL
LIN {X 0,Y 328.846,Z 703.008,A -85,B 0,C 180,E1 -23291.76,E2 -23291.76} C_VEL
LIN {X 0,Y 333.832,Z 706.246,A -85,B 0,C 180,E1 -23293.543,E2 -23293.543} C_VEL
LIN {X 0,Y 339.057,Z 709.367,A -85,B 0,C 180,E1 -23295.598,E2 -23295.598} C_VEL
LIN {X 0,Y 341.85,Z 711.457,A -85,B 0,C 180,E1 -23296.93,E2 -23296.93} C_VEL
LIN {X 0,Y 344.455,Z 713.357,A -85,B 0,C 180,E1 -23298.333,E2 -23298.333} C_VEL
LIN {X 0,Y 348.482,Z 715.79,A -85,B 0,C 180,E1 -23300.716,E2 -23300.716} C_VEL
LIN {X 0,Y 350.265,Z 716.703,A -85,B 0,C 180,E1 -23301.926,E2 -23301.926} C_VEL
LIN {X 0,Y 351.768,Z 717.437,A -85,B 0,C 180,E1 -23303.115,E2 -23303.115} C_VEL
LIN {X 0,Y 354.041,Z 718.452,A -85,B 0,C 180,E1 -23305.446,E2 -23305.446} C_VEL
LIN {X 0,Y 354.893,Z 718.702,A -85,B 0,C 180,E1 -23306.594,E2 -23306.594} C_VEL
LIN {X 0,Y 355.752,Z 719.143,A -85,B 0,C 180,E1 -23308.868,E2 -23308.868} C_VEL
LIN {X 0,Y 355.932,Z 719.095,A -85,B 0,C 180,E1 -23310,E2 -23310} C_VEL
LIN {X 0,Y 355.447,Z 718.955,A -85,B 0,C 180,E1 -23312.266,E2 -23312.266} C_VEL
LIN {X 0,Y 354.888,Z 718.711,A -85,B 0,C 180,E1 -23313.406,E2 -23313.406} C_VEL
LIN {X 0,Y 353.01,Z 718.005,A -85,B 0,C 180,E1 -23315.713,E2 -23315.713} C_VEL
LIN {X 0,Y 351.752,Z 717.429,A -85,B 0,C 180,E1 -23316.885,E2 -23316.885} C_VEL
LIN {X 0,Y 348.755,Z 715.918,A -85,B 0,C 180,E1 -23319.098,E2 -23319.098} C_VEL
LIN {X 0,Y 346.525,Z 714.602,A -85,B 0,C 180,E1 -23320.517,E2 -23320.517} C_VEL
LIN {X 0,Y 344.278,Z 713.197,A -85,B 0,C 180,E1 -23321.779,E2 -23321.779} C_VEL
LIN {X 0,Y 340.23,Z 710.188,A -85,B 0,C 180,E1 -23323.869,E2 -23323.869} C_VEL
LIN {X 0,Y 335.631,Z 707.284,A -85,B 0,C 180,E1 -23325.796,E2 -23325.796} C_VEL
LIN {X 0,Y 331.351,Z 704.72,A -85,B 0,C 180,E1 -23327.361,E2 -23327.361} C_VEL
LIN {X 0,Y 325.779,Z 700.768,A -85,B 0,C 180,E1 -23329.295,E2 -23329.295} C_VEL
LIN {X 0,Y 322.355,Z 698.203,A -85,B 0,C 180,E1 -23330.415,E2 -23330.415} C_VEL
LIN {X 0,Y 316.065,Z 694.044,A -85,B 0,C 180,E1 -23332.21,E2 -23332.21} C_VEL
LIN {X 0,Y 308.395,Z 688.315,A -85,B 0,C 180,E1 -23334.28,E2 -23334.28} C_VEL
LIN {X 0,Y 301.103,Z 683.141,A -85,B 0,C 180,E1 -23336.026,E2 -23336.026} C_VEL
LIN {X 0,Y 293.636,Z 677.469,A -85,B 0,C 180,E1 -23337.68,E2 -23337.68} C_VEL
LIN {X 0,Y 285.907,Z 671.688,A -85,B 0,C 180,E1 -23339.235,E2 -23339.235} C_VEL
LIN {X 0,Y 270.949,Z 659.782,A -85,B 0,C 180,E1 -23342.109,E2 -23342.109} C_VEL
LIN {X 0,Y 261.311,Z 651.483,A -85,B 0,C 180,E1 -23344.062,E2 -23344.062} C_VEL
LIN {X 0,Y 250.816,Z 641.462,A -85,B 0,C 180,E1 -23346.297,E2 -23346.297} C_VEL
LIN {X 0,Y 237.286,Z 627.179,A -85,B 0,C 180,E1 -23349.346,E2 -23349.346} C_VEL
LIN {X 0,Y 226.615,Z 613.789,A -85,B 0,C 180,E1 -23352.171,E2 -23352.171} C_VEL
LIN {X 0,Y 217.193,Z 598.888,A -85,B 0,C 180,E1 -23355.164,E2 -23355.164} C_VEL
LIN {X 0,Y 206.904,Z 578.424,A -85,B 0,C 180,E1 -23359.185,E2 -23359.185} C_VEL
LIN {X 0,Y 200.746,Z 567.456,A -85,B 0,C 180,E1 -23361.901,E2 -23361.901} C_VEL
LIN {X 0,Y 194.66,Z 557.75,A -85,B 0,C 180,E1 -23364.873,E2 -23364.873} C_VEL
LIN {X 0,Y 188.9,Z 549.556,A -85,B 0,C 180,E1 -23368.034,E2 -23368.034} C_VEL
LIN {X 0,Y 185.813,Z 545.35,A -85,B 0,C 180,E1 -23369.925,E2 -23369.925} C_VEL
LIN {X 0,Y 182.525,Z 540.966,A -85,B 0,C 180,E1 -23372.135,E2 -23372.135} C_VEL
LIN {X 0,Y 179.895,Z 537.833,A -85,B 0,C 180,E1 -23374.058,E2 -23374.058} C_VEL
LIN {X 0,Y 178.762,Z 536.141,A -85,B 0,C 180,E1 -23374.98,E2 -23374.98} C_VEL
LIN {X 0,Y 176.077,Z 533.503,A -85,B 0,C 180,E1 -23377.215,E2 -23377.215} C_VEL
LIN {X 0,Y 174.538,Z 530.879,A -85,B 0,C 180,E1 -23378.754,E2 -23378.754} C_VEL
LIN {X 0,Y 171.95,Z 528.88,A -85,B 0,C 180,E1 -23381.38,E2 -23381.38} C_VEL
LIN {X 0,Y 169.909,Z 525.399,A -85,B 0,C 180,E1 -23384.097,E2 -23384.097} C_VEL
LIN {X 0,Y 166.531,Z 522.953,A -85,B 0,C 180,E1 -23389.536,E2 -23389.536} C_VEL
LIN {X 0,Y 164.937,Z 519.934,A -85,B 0,C 180,E1 -23395.112,E2 -23395.112} C_VEL
LIN {X 0,Y 165.155,Z 519.194,A -85,B 0,C 180,E1 -23398.782,E2 -23398.782} C_VEL
LIN {X 0,Y 165.156,Z 519.225,A -85,B 0,C 180,E1 -23401.22,E2 -23401.22} C_VEL
LIN {X 0,Y 165.011,Z 520.18,A -85,B 0,C 180,E1 -23405.194,E2 -23405.194} C_VEL
LIN {X 0,Y 168.5,Z 524.621,A -85,B 0,C 180,E1 -23413.57,E2 -23413.57} C_VEL
LIN {X 0,Y 170.07,Z 525.615,A -85,B 0,C 180,E1 -23415.736,E2 -23415.736} C_VEL
LIN {X 0,Y 171.542,Z 528.34,A -85,B 0,C 180,E1 -23417.742,E2 -23417.742} C_VEL
LIN {X 0,Y 174.085,Z 530.628,A -85,B 0,C 180,E1 -23420.434,E2 -23420.434} C_VEL
LIN {X 0,Y 174.824,Z 531.278,A -85,B 0,C 180,E1 -23421.14,E2 -23421.14} C_VEL
LIN {X 0,Y 176.716,Z 534.345,A -85,B 0,C 180,E1 -23422.971,E2 -23422.971} C_VEL
LIN {X 0,Y 179.198,Z 536.627,A -85,B 0,C 180,E1 -23424.972,E2 -23424.972} C_VEL
LIN {X 0,Y 181.849,Z 540.319,A -85,B 0,C 180,E1 -23427.009,E2 -23427.009} C_VEL
LIN {X 0,Y 183.285,Z 541.947,A -85,B 0,C 180,E1 -23428.002,E2 -23428.002} C_VEL
LIN {X 0,Y 186.978,Z 546.932,A -85,B 0,C 180,E1 -23430.416,E2 -23430.416} C_VEL
LIN {X 0,Y 190.271,Z 551.507,A -85,B 0,C 180,E1 -23432.368,E2 -23432.368} C_VEL
LIN {X 0,Y 194.67,Z 559.25,A -85,B 0,C 180,E1 -23434.833,E2 -23434.833} C_VEL
LIN {X 0,Y 200.446,Z 570.575,A -85,B 0,C 180,E1 -23437.774,E2 -23437.774} C_VEL
LIN {X 0,Y 205.93,Z 582.97,A -85,B 0,C 180,E1 -23440.344,E2 -23440.344} C_VEL
LIN {X 0,Y 210.148,Z 594.05,A -85,B 0,C 180,E1 -23442.224,E2 -23442.224} C_VEL
LIN {X 0,Y 206.356,Z 650.4,A -85,B 0,C 180,E1 -23443.958,E2 -23443.958} C_VEL
LIN {X 0,Y 204.966,Z 661.661,A -85,B 0,C 180,E1 -23444.47,E2 -23444.47} C_VEL
LIN {X 0,Y 203.329,Z 671.289,A -85,B 0,C 180,E1 -23445.057,E2 -23445.057} C_VEL
LIN {X 0,Y 200.857,Z 682.437,A -85,B 0,C 180,E1 -23445.94,E2 -23445.94} C_VEL
LIN {X 0,Y 198.215,Z 692.403,A -85,B 0,C 180,E1 -23446.959,E2 -23446.959} C_VEL
LIN {X 0,Y 195.171,Z 702.319,A -85,B 0,C 180,E1 -23448.229,E2 -23448.229} C_VEL
LIN {X 0,Y 191.737,Z 712.038,A -85,B 0,C 180,E1 -23449.758,E2 -23449.758} C_VEL
LIN {X 0,Y 188.002,Z 721.708,A -85,B 0,C 180,E1 -23451.658,E2 -23451.658} C_VEL
LIN {X 0,Y 184.255,Z 730.475,A -85,B 0,C 180,E1 -23453.758,E2 -23453.758} C_VEL
LIN {X 0,Y 180.995,Z 737.446,A -85,B 0,C 180,E1 -23455.735,E2 -23455.735} C_VEL
LIN {X 0,Y 177.206,Z 744.965,A -85,B 0,C 180,E1 -23458.299,E2 -23458.299} C_VEL
LIN {X 0,Y 173.258,Z 752.576,A -85,B 0,C 180,E1 -23461.536,E2 -23461.536} C_VEL
LIN {X 0,Y 170.387,Z 757.979,A -85,B 0,C 180,E1 -23464.336,E2 -23464.336} C_VEL
LIN {X 0,Y 167.558,Z 763.416,A -85,B 0,C 180,E1 -23467.822,E2 -23467.822} C_VEL
LIN {X 0,Y 165.322,Z 767.867,A -85,B 0,C 180,E1 -23471.408,E2 -23471.408} C_VEL
LIN {X 0,Y 163.553,Z 771.416,A -85,B 0,C 180,E1 -23475.059,E2 -23475.059} C_VEL
LIN {X 0,Y 162.792,Z 773.363,A -85,B 0,C 180,E1 -23477.534,E2 -23477.534} C_VEL
LIN {X 0,Y 161.882,Z 776.218,A -85,B 0,C 180,E1 -23482.989,E2 -23482.989} C_VEL
LIN {X 0,Y 161.799,Z 777.367,A -85,B 0,C 180,E1 -23487.511,E2 -23487.511} C_VEL
LIN {X 0,Y 161.9,Z 777.624,A -85,B 0,C 180,E1 -23490,E2 -23490} C_VEL
LIN {X 0,Y 161.758,Z 777.119,A -85,B 0,C 180,E1 -23493.78,E2 -23493.78} C_VEL
LIN {X 0,Y 161.141,Z 776.608,A -85,B 0,C 180,E1 -23495.854,E2 -23495.854} C_VEL
LIN {X 0,Y 159.71,Z 775.897,A -85,B 0,C 180,E1 -23497.898,E2 -23497.898} C_VEL
LIN {X 0,Y 156.682,Z 773.768,A -85,B 0,C 180,E1 -23502.022,E2 -23502.022} C_VEL
LIN {X 0,Y 156.22,Z 772.339,A -85,B 0,C 180,E1 -23504.134,E2 -23504.134} C_VEL
LIN {X 0,Y 156.369,Z 771.807,A -85,B 0,C 180,E1 -23504.834,E2 -23504.834} C_VEL
LIN {X 0,Y 157.864,Z 768.936,A -85,B 0,C 180,E1 -23508.157,E2 -23508.157} C_VEL
LIN {X 0,Y 160.098,Z 764.798,A -85,B 0,C 180,E1 -23511.908,E2 -23511.908} C_VEL
LIN {X 0,Y 162.878,Z 759.693,A -85,B 0,C 180,E1 -23515.561,E2 -23515.561} C_VEL
LIN {X 0,Y 166.384,Z 753.515,A -85,B 0,C 180,E1 -23519.061,E2 -23519.061} C_VEL
LIN {X 0,Y 169.711,Z 747.44,A -85,B 0,C 180,E1 -23521.869,E2 -23521.869} C_VEL
LIN {X 0,Y 173.518,Z 740.369,A -85,B 0,C 180,E1 -23524.543,E2 -23524.543} C_VEL
LIN {X 0,Y 177.744,Z 732.096,A -85,B 0,C 180,E1 -23527.083,E2 -23527.083} C_VEL
LIN {X 0,Y 181.902,Z 722.922,A -85,B 0,C 180,E1 -23529.4,E2 -23529.4} C_VEL
LIN {X 0,Y 185.426,Z 714.32,A -85,B 0,C 180,E1 -23531.188,E2 -23531.188} C_VEL
LIN {X 0,Y 188.922,Z 705.049,A -85,B 0,C 180,E1 -23532.757,E2 -23532.757} C_VEL
LIN {X 0,Y 192.015,Z 695.711,A -85,B 0,C 180,E1 -23534.06,E2 -23534.06} C_VEL
LIN {X 0,Y 194.996,Z 685.458,A -85,B 0,C 180,E1 -23535.199,E2 -23535.199} C_VEL
LIN {X 0,Y 197.768,Z 673.809,A -85,B 0,C 180,E1 -23536.205,E2 -23536.205} C_VEL
LIN {X 0,Y 199.75,Z 663.286,A -85,B 0,C 180,E1 -23536.891,E2 -23536.891} C_VEL
LIN {X 0,Y 201.346,Z 651.618,A -85,B 0,C 180,E1 -23537.431,E2 -23537.431} C_VEL
LIN {X 0,Y 203.237,Z 626.995,A -85,B 0,C 180,E1 -23538.22,E2 -23538.22} C_VEL
LIN {X 0,Y 205.291,Z 596.319,A -85,B 0,C 180,E1 -23539.163,E2 -23539.163} C_VEL
LIN {X 0,Y 200.857,Z 584.651,A -85,B 0,C 180,E1 -23541.284,E2 -23541.284} C_VEL
LIN {X 0,Y 196.018,Z 573.669,A -85,B 0,C 180,E1 -23543.729,E2 -23543.729} C_VEL
LIN {X 0,Y 190.691,Z 562.992,A -85,B 0,C 180,E1 -23546.66,E2 -23546.66} C_VEL
LIN {X 0,Y 186.8,Z 556.098,A -85,B 0,C 180,E1 -23549.004,E2 -23549.004} C_VEL
LIN {X 0,Y 182.78,Z 550.693,A -85,B 0,C 180,E1 -23551.583,E2 -23551.583} C_VEL
LIN {X 0,Y 180.296,Z 547.207,A -85,B 0,C 180,E1 -23553.366,E2 -23553.366} C_VEL
LIN {X 0,Y 177.339,Z 543.309,A -85,B 0,C 180,E1 -23555.691,E2 -23555.691} C_VEL
LIN {X 0,Y 173.764,Z 539.223,A -85,B 0,C 180,E1 -23558.871,E2 -23558.871} C_VEL
LIN {X 0,Y 172.798,Z 537.529,A -85,B 0,C 180,E1 -23559.905,E2 -23559.905} C_VEL
LIN {X 0,Y 170.091,Z 535.049,A -85,B 0,C 180,E1 -23562.877,E2 -23562.877} C_VEL
LIN {X 0,Y 168.425,Z 532.102,A -85,B 0,C 180,E1 -23565.268,E2 -23565.268} C_VEL
LIN {X 0,Y 165.513,Z 529.905,A -85,B 0,C 180,E1 -23570.22,E2 -23570.22} C_VEL
LIN {X 0,Y 163.834,Z 526.777,A -85,B 0,C 180,E1 -23576.002,E2 -23576.002} C_VEL
LIN {X 0,Y 163.497,Z 525.956,A -85,B 0,C 180,E1 -23579.999,E2 -23579.999} C_VEL
LIN {X 0,Y 163.867,Z 526.896,A -85,B 0,C 180,E1 -23584.611,E2 -23584.611} C_VEL
LIN {X 0,Y 166.849,Z 531.261,A -85,B 0,C 180,E1 -23592.775,E2 -23592.775} C_VEL
LIN {X 0,Y 168.623,Z 532.311,A -85,B 0,C 180,E1 -23595.407,E2 -23595.407} C_VEL
LIN {X 0,Y 170.603,Z 535.732,A -85,B 0,C 180,E1 -23598.151,E2 -23598.151} C_VEL
LIN {X 0,Y 173.136,Z 537.999,A -85,B 0,C 180,E1 -23600.842,E2 -23600.842} C_VEL
LIN {X 0,Y 175.534,Z 541.506,A -85,B 0,C 180,E1 -23603.191,E2 -23603.191} C_VEL
LIN {X 0,Y 177.323,Z 543.247,A -85,B 0,C 180,E1 -23604.684,E2 -23604.684} C_VEL
LIN {X 0,Y 180.021,Z 546.962,A -85,B 0,C 180,E1 -23606.832,E2 -23606.832} C_VEL
LIN {X 0,Y 181.248,Z 548.554,A -85,B 0,C 180,E1 -23607.729,E2 -23607.729} C_VEL
LIN {X 0,Y 184.82,Z 553.441,A -85,B 0,C 180,E1 -23610.157,E2 -23610.157} C_VEL
LIN {X 0,Y 189.85,Z 560.613,A -85,B 0,C 180,E1 -23613.186,E2 -23613.186} C_VEL
LIN {X 0,Y 195.765,Z 569.988,A -85,B 0,C 180,E1 -23616.339,E2 -23616.339} C_VEL
LIN {X 0,Y 201.356,Z 579.889,A -85,B 0,C 180,E1 -23619.019,E2 -23619.019} C_VEL
LIN {X 0,Y 206.562,Z 590.258,A -85,B 0,C 180,E1 -23621.32,E2 -23621.32} C_VEL
LIN {X 0,Y 213.91,Z 605.042,A -85,B 0,C 180,E1 -23624.23,E2 -23624.23} C_VEL
LIN {X 0,Y 222.739,Z 619.076,A -85,B 0,C 180,E1 -23627.142,E2 -23627.142} C_VEL
LIN {X 0,Y 234.28,Z 633.701,A -85,B 0,C 180,E1 -23630.3,E2 -23630.3} C_VEL
LIN {X 0,Y 246.702,Z 646.954,A -85,B 0,C 180,E1 -23633.287,E2 -23633.287} C_VEL
LIN {X 0,Y 258.531,Z 658.461,A -85,B 0,C 180,E1 -23636.007,E2 -23636.007} C_VEL
LIN {X 0,Y 272.016,Z 669.868,A -85,B 0,C 180,E1 -23638.887,E2 -23638.887} C_VEL
LIN {X 0,Y 284.296,Z 679.377,A -85,B 0,C 180,E1 -23641.35,E2 -23641.35} C_VEL
LIN {X 0,Y 293.794,Z 686.553,A -85,B 0,C 180,E1 -23643.343,E2 -23643.343} C_VEL
LIN {X 0,Y 301.872,Z 692.384,A -85,B 0,C 180,E1 -23645.225,E2 -23645.225} C_VEL
LIN {X 0,Y 309.03,Z 697.729,A -85,B 0,C 180,E1 -23647.08,E2 -23647.08} C_VEL
LIN {X 0,Y 316.546,Z 702.908,A -85,B 0,C 180,E1 -23649.193,E2 -23649.193} C_VEL
LIN {X 0,Y 321.876,Z 706.709,A -85,B 0,C 180,E1 -23650.882,E2 -23650.882} C_VEL
LIN {X 0,Y 326.434,Z 709.933,A -85,B 0,C 180,E1 -23652.458,E2 -23652.458} C_VEL
LIN {X 0,Y 332.46,Z 713.61,A -85,B 0,C 180,E1 -23654.667,E2 -23654.667} C_VEL
LIN {X 0,Y 335.422,Z 715.467,A -85,B 0,C 180,E1 -23655.929,E2 -23655.929} C_VEL
LIN {X 0,Y 339.596,Z 718.603,A -85,B 0,C 180,E1 -23658.057,E2 -23658.057} C_VEL
LIN {X 0,Y 342.72,Z 720.57,A -85,B 0,C 180,E1 -23659.834,E2 -23659.834} C_VEL
LIN {X 0,Y 345.75,Z 722.238,A -85,B 0,C 180,E1 -23661.82,E2 -23661.82} C_VEL
LIN {X 0,Y 347.332,Z 722.994,A -85,B 0,C 180,E1 -23663.027,E2 -23663.027} C_VEL
LIN {X 0,Y 348.626,Z 723.64,A -85,B 0,C 180,E1 -23664.215,E2 -23664.215} C_VEL
LIN {X 0,Y 350.58,Z 724.356,A -85,B 0,C 180,E1 -23666.552,E2 -23666.552} C_VEL
LIN {X 0,Y 351.48,Z 724.789,A -85,B 0,C 180,E1 -23668.854,E2 -23668.854} C_VEL
LIN {X 0,Y 351.662,Z 724.755,A -85,B 0,C 180,E1 -23670,E2 -23670} C_VEL
LIN {X 0,Y 351.156,Z 724.616,A -85,B 0,C 180,E1 -23672.294,E2 -23672.294} C_VEL
LIN {X 0,Y 350.575,Z 724.37,A -85,B 0,C 180,E1 -23673.448,E2 -23673.448} C_VEL
LIN {X 0,Y 348.637,Z 723.618,A -85,B 0,C 180,E1 -23675.785,E2 -23675.785} C_VEL
LIN {X 0,Y 347.075,Z 722.893,A -85,B 0,C 180,E1 -23677.162,E2 -23677.162} C_VEL
LIN {X 0,Y 343.928,Z 721.257,A -85,B 0,C 180,E1 -23679.408,E2 -23679.408} C_VEL
LIN {X 0,Y 341.917,Z 720.063,A -85,B 0,C 180,E1 -23680.66,E2 -23680.66} C_VEL
LIN {X 0,Y 338.43,Z 717.733,A -85,B 0,C 180,E1 -23682.576,E2 -23682.576} C_VEL
LIN {X 0,Y 334.133,Z 714.641,A -85,B 0,C 180,E1 -23684.641,E2 -23684.641} C_VEL
LIN {X 0,Y 329.658,Z 711.942,A -85,B 0,C 180,E1 -23686.394,E2 -23686.394} C_VEL
LIN {X 0,Y 325.136,Z 709.053,A -85,B 0,C 180,E1 -23687.997,E2 -23687.997} C_VEL
LIN {X 0,Y 320.654,Z 705.75,A -85,B 0,C 180,E1 -23689.533,E2 -23689.533} C_VEL
LIN {X 0,Y 314.366,Z 701.42,A -85,B 0,C 180,E1 -23691.438,E2 -23691.438} C_VEL
LIN {X 0,Y 306.686,Z 695.943,A -85,B 0,C 180,E1 -23693.563,E2 -23693.563} C_VEL
LIN {X 0,Y 299.408,Z 690.727,A -85,B 0,C 180,E1 -23695.352,E2 -23695.352} C_VEL
LIN {X 0,Y 291.994,Z 685.056,A -85,B 0,C 180,E1 -23697.059,E2 -23697.059} C_VEL
LIN {X 0,Y 282.99,Z 678.38,A -85,B 0,C 180,E1 -23698.906,E2 -23698.906} C_VEL
LIN {X 0,Y 267.455,Z 666.068,A -85,B 0,C 180,E1 -23702.067,E2 -23702.067} C_VEL
LIN {X 0,Y 257.602,Z 657.53,A -85,B 0,C 180,E1 -23704.21,E2 -23704.21} C_VEL
LIN {X 0,Y 246.842,Z 647.106,A -85,B 0,C 180,E1 -23706.68,E2 -23706.68} C_VEL
LIN {X 0,Y 234.608,Z 634.057,A -85,B 0,C 180,E1 -23709.619,E2 -23709.619} C_VEL
LIN {X 0,Y 224.108,Z 620.917,A -85,B 0,C 180,E1 -23712.453,E2 -23712.453} C_VEL
LIN {X 0,Y 216.943,Z 610.181,A -85,B 0,C 180,E1 -23714.711,E2 -23714.711} C_VEL
LIN {X 0,Y 210.317,Z 598.228,A -85,B 0,C 180,E1 -23717.127,E2 -23717.127} C_VEL
LIN {X 0,Y 203.188,Z 583.353,A -85,B 0,C 180,E1 -23720.155,E2 -23720.155} C_VEL
LIN {X 0,Y 197.214,Z 572.452,A -85,B 0,C 180,E1 -23722.941,E2 -23722.941} C_VEL
LIN {X 0,Y 191.562,Z 563.203,A -85,B 0,C 180,E1 -23725.863,E2 -23725.863} C_VEL
LIN {X 0,Y 185.996,Z 555.139,A -85,B 0,C 180,E1 -23729.094,E2 -23729.094} C_VEL
LIN {X 0,Y 183.261,Z 551.265,A -85,B 0,C 180,E1 -23730.871,E2 -23730.871} C_VEL
LIN {X 0,Y 180.2,Z 547.136,A -85,B 0,C 180,E1 -23733.04,E2 -23733.04} C_VEL
LIN {X 0,Y 177.372,Z 543.377,A -85,B 0,C 180,E1 -23735.269,E2 -23735.269} C_VEL
LIN {X 0,Y 176.272,Z 542.189,A -85,B 0,C 180,E1 -23736.182,E2 -23736.182} C_VEL
LIN {X 0,Y 173.671,Z 539.021,A -85,B 0,C 180,E1 -23738.58,E2 -23738.58} C_VEL
LIN {X 0,Y 172.758,Z 537.525,A -85,B 0,C 180,E1 -23739.549,E2 -23739.549} C_VEL
LIN {X 0,Y 170.14,Z 535.136,A -85,B 0,C 180,E1 -23742.42,E2 -23742.42} C_VEL
LIN {X 0,Y 168.425,Z 532.058,A -85,B 0,C 180,E1 -23744.884,E2 -23744.884} C_VEL
LIN {X 0,Y 165.753,Z 530.234,A -85,B 0,C 180,E1 -23749.291,E2 -23749.291} C_VEL
LIN {X 0,Y 163.865,Z 526.91,A -85,B 0,C 180,E1 -23755.389,E2 -23755.389} C_VEL
LIN {X 0,Y 163.504,Z 526.103,A -85,B 0,C 180,E1 -23758.77,E2 -23758.77} C_VEL
LIN {X 0,Y 163.625,Z 526.333,A -85,B 0,C 180,E1 -23762.463,E2 -23762.463} C_VEL
LIN {X 0,Y 164.484,Z 528.175,A -85,B 0,C 180,E1 -23766.903,E2 -23766.903} C_VEL
LIN {X 0,Y 167.268,Z 531.491,A -85,B 0,C 180,E1 -23773.053,E2 -23773.053} C_VEL
LIN {X 0,Y 168.628,Z 532.319,A -85,B 0,C 180,E1 -23775.023,E2 -23775.023} C_VEL
LIN {X 0,Y 170.493,Z 535.575,A -85,B 0,C 180,E1 -23777.622,E2 -23777.622} C_VEL
LIN {X 0,Y 173.158,Z 538.055,A -85,B 0,C 180,E1 -23780.475,E2 -23780.475} C_VEL
LIN {X 0,Y 175.403,Z 541.385,A -85,B 0,C 180,E1 -23782.685,E2 -23782.685} C_VEL
LIN {X 0,Y 177.339,Z 543.311,A -85,B 0,C 180,E1 -23784.309,E2 -23784.309} C_VEL
LIN {X 0,Y 180.294,Z 547.22,A -85,B 0,C 180,E1 -23786.634,E2 -23786.634} C_VEL
LIN {X 0,Y 184.744,Z 553.369,A -85,B 0,C 180,E1 -23789.719,E2 -23789.719} C_VEL
LIN {X 0,Y 187.678,Z 557.563,A -85,B 0,C 180,E1 -23791.541,E2 -23791.541} C_VEL
LIN {X 0,Y 192.844,Z 567.135,A -85,B 0,C 180,E1 -23794.559,E2 -23794.559} C_VEL
LIN {X 0,Y 198.201,Z 578.439,A -85,B 0,C 180,E1 -23797.395,E2 -23797.395} C_VEL
LIN {X 0,Y 203.333,Z 590.951,A -85,B 0,C 180,E1 -23799.912,E2 -23799.912} C_VEL
LIN {X 0,Y 205.287,Z 596.287,A -85,B 0,C 180,E1 -23800.834,E2 -23800.834} C_VEL
LIN {X 0,Y 201.43,Z 650.929,A -85,B 0,C 180,E1 -23802.536,E2 -23802.536} C_VEL
LIN {X 0,Y 199.775,Z 663.287,A -85,B 0,C 180,E1 -23803.117,E2 -23803.117} C_VEL
LIN {X 0,Y 197.537,Z 675.171,A -85,B 0,C 180,E1 -23803.909,E2 -23803.909} C_VEL
LIN {X 0,Y 194.16,Z 688.643,A -85,B 0,C 180,E1 -23805.104,E2 -23805.104} C_VEL
LIN {X 0,Y 189.927,Z 702.12,A -85,B 0,C 180,E1 -23806.8,E2 -23806.8} C_VEL
LIN {X 0,Y 186.368,Z 711.839,A -85,B 0,C 180,E1 -23808.346,E2 -23808.346} C_VEL
LIN {X 0,Y 183.113,Z 719.995,A -85,B 0,C 180,E1 -23809.926,E2 -23809.926} C_VEL
LIN {X 0,Y 179.425,Z 728.457,A -85,B 0,C 180,E1 -23811.909,E2 -23811.909} C_VEL
LIN {X 0,Y 175.157,Z 737.247,A -85,B 0,C 180,E1 -23814.424,E2 -23814.424} C_VEL
LIN {X 0,Y 171.175,Z 744.766,A -85,B 0,C 180,E1 -23817.044,E2 -23817.044} C_VEL
LIN {X 0,Y 167.006,Z 752.377,A -85,B 0,C 180,E1 -23820.366,E2 -23820.366} C_VEL
LIN {X 0,Y 163.982,Z 757.78,A -85,B 0,C 180,E1 -23823.256,E2 -23823.256} C_VEL
LIN {X 0,Y 160.924,Z 763.216,A -85,B 0,C 180,E1 -23826.856,E2 -23826.856} C_VEL
LIN {X 0,Y 158.563,Z 767.668,A -85,B 0,C 180,E1 -23830.585,E2 -23830.585} C_VEL
LIN {X 0,Y 156.655,Z 771.217,A -85,B 0,C 180,E1 -23834.385,E2 -23834.385} C_VEL
LIN {X 0,Y 155.826,Z 773.164,A -85,B 0,C 180,E1 -23836.968,E2 -23836.968} C_VEL
LIN {X 0,Y 154.865,Z 775.864,A -85,B 0,C 180,E1 -23842.175,E2 -23842.175} C_VEL
LIN {X 0,Y 154.7,Z 777.169,A -85,B 0,C 180,E1 -23847.396,E2 -23847.396} C_VEL
LIN {X 0,Y 154.799,Z 777.426,A -85,B 0,C 180,E1 -23850,E2 -23850} C_VEL
LIN {X 0,Y 154.71,Z 776.689,A -85,B 0,C 180,E1 -23855.213,E2 -23855.213} C_VEL
LIN {X 0,Y 154.865,Z 775.864,A -85,B 0,C 180,E1 -23857.825,E2 -23857.825} C_VEL
LIN {X 0,Y 155.826,Z 773.164,A -85,B 0,C 180,E1 -23863.032,E2 -23863.032} C_VEL
LIN {X 0,Y 156.369,Z 771.807,A -85,B 0,C 180,E1 -23864.834,E2 -23864.834} C_VEL
LIN {X 0,Y 156.509,Z 770.223,A -85,B 0,C 180,E1 -23866.92,E2 -23866.92} C_VEL
LIN {X 0,Y 155.35,Z 767.188,A -85,B 0,C 180,E1 -23870.379,E2 -23870.379} C_VEL
LIN {X 0,Y 154.696,Z 763.574,A -85,B 0,C 180,E1 -23873.79,E2 -23873.79} C_VEL
LIN {X 0,Y 155.598,Z 760.978,A -85,B 0,C 180,E1 -23875.724,E2 -23875.724} C_VEL
LIN {X 0,Y 159.504,Z 754.453,A -85,B 0,C 180,E1 -23879.715,E2 -23879.715} C_VEL
LIN {X 0,Y 163.68,Z 747.241,A -85,B 0,C 180,E1 -23883.191,E2 -23883.191} C_VEL
LIN {X 0,Y 167.68,Z 740.17,A -85,B 0,C 180,E1 -23885.928,E2 -23885.928} C_VEL
LIN {X 0,Y 171.185,Z 733.714,A -85,B 0,C 180,E1 -23888.011,E2 -23888.011} C_VEL
LIN {X 0,Y 176.122,Z 723.473,A -85,B 0,C 180,E1 -23890.695,E2 -23890.695} C_VEL
LIN {X 0,Y 179.622,Z 715.361,A -85,B 0,C 180,E1 -23892.448,E2 -23892.448} C_VEL
LIN {X 0,Y 183.224,Z 706.314,A -85,B 0,C 180,E1 -23894.044,E2 -23894.044} C_VEL
LIN {X 0,Y 186.966,Z 695.512,A -85,B 0,C 180,E1 -23895.577,E2 -23895.577} C_VEL
LIN {X 0,Y 190.056,Z 685.26,A -85,B 0,C 180,E1 -23896.719,E2 -23896.719} C_VEL
LIN {X 0,Y 192.931,Z 673.611,A -85,B 0,C 180,E1 -23897.724,E2 -23897.724} C_VEL
LIN {X 0,Y 195.11,Z 662.176,A -85,B 0,C 180,E1 -23898.464,E2 -23898.464} C_VEL
LIN {X 0,Y 196.604,Z 651.288,A -85,B 0,C 180,E1 -23898.967,E2 -23898.967} C_VEL
LIN {X 0,Y 198.482,Z 628.354,A -85,B 0,C 180,E1 -23899.694,E2 -23899.694} C_VEL
LIN {X 0,Y 200.523,Z 598.482,A -85,B 0,C 180,E1 -23900.634,E2 -23900.634} C_VEL
LIN {X 0,Y 196.046,Z 586.762,A -85,B 0,C 180,E1 -23902.935,E2 -23902.935} C_VEL
LIN {X 0,Y 191.846,Z 577.071,A -85,B 0,C 180,E1 -23905.232,E2 -23905.232} C_VEL
LIN {X 0,Y 187.21,Z 567.618,A -85,B 0,C 180,E1 -23907.976,E2 -23907.976} C_VEL
LIN {X 0,Y 184.161,Z 561.951,A -85,B 0,C 180,E1 -23909.941,E2 -23909.941} C_VEL
LIN {X 0,Y 180.345,Z 556.698,A -85,B 0,C 180,E1 -23912.527,E2 -23912.527} C_VEL
LIN {X 0,Y 177.883,Z 553.193,A -85,B 0,C 180,E1 -23914.396,E2 -23914.396} C_VEL
LIN {X 0,Y 174.717,Z 548.964,A -85,B 0,C 180,E1 -23917.064,E2 -23917.064} C_VEL
LIN {X 0,Y 171.882,Z 545.478,A -85,B 0,C 180,E1 -23919.793,E2 -23919.793} C_VEL
LIN {X 0,Y 171.171,Z 544.225,A -85,B 0,C 180,E1 -23920.596,E2 -23920.596} C_VEL
LIN {X 0,Y 168.553,Z 541.601,A -85,B 0,C 180,E1 -23923.652,E2 -23923.652} C_VEL
LIN {X 0,Y 167.215,Z 538.997,A -85,B 0,C 180,E1 -23925.703,E2 -23925.703} C_VEL
LIN {X 0,Y 164.392,Z 536.718,A -85,B 0,C 180,E1 -23930.774,E2 -23930.774} C_VEL
LIN {X 0,Y 162.872,Z 533.65,A -85,B 0,C 180,E1 -23936.597,E2 -23936.597} C_VEL
LIN {X 0,Y 162.631,Z 533.007,A -85,B 0,C 180,E1 -23939.999,E2 -23939.999} C_VEL
LIN {X 0,Y 162.995,Z 534.02,A -85,B 0,C 180,E1 -23944.636,E2 -23944.636} C_VEL
LIN {X 0,Y 166.003,Z 538.324,A -85,B 0,C 180,E1 -23952.841,E2 -23952.841} C_VEL
LIN {X 0,Y 167.266,Z 539.154,A -85,B 0,C 180,E1 -23954.783,E2 -23954.783} C_VEL
LIN {X 0,Y 169.506,Z 542.826,A -85,B 0,C 180,E1 -23957.96,E2 -23957.96} C_VEL
LIN {X 0,Y 171.491,Z 544.688,A -85,B 0,C 180,E1 -23960.151,E2 -23960.151} C_VEL
LIN {X 0,Y 174.022,Z 548.3,A -85,B 0,C 180,E1 -23962.716,E2 -23962.716} C_VEL
LIN {X 0,Y 175.494,Z 549.929,A -85,B 0,C 180,E1 -23964.01,E2 -23964.01} C_VEL
LIN {X 0,Y 179.144,Z 554.973,A -85,B 0,C 180,E1 -23966.974,E2 -23966.974} C_VEL
LIN {X 0,Y 182.483,Z 559.663,A -85,B 0,C 180,E1 -23969.355,E2 -23969.355} C_VEL
LIN {X 0,Y 187.548,Z 567.188,A -85,B 0,C 180,E1 -23972.55,E2 -23972.55} C_VEL
LIN {X 0,Y 192.954,Z 576.048,A -85,B 0,C 180,E1 -23975.564,E2 -23975.564} C_VEL
LIN {X 0,Y 198.636,Z 586.537,A -85,B 0,C 180,E1 -23978.416,E2 -23978.416} C_VEL
LIN {X 0,Y 203.332,Z 596.469,A -85,B 0,C 180,E1 -23980.599,E2 -23980.599} C_VEL
LIN {X 0,Y 211.054,Z 611.943,A -85,B 0,C 180,E1 -23983.757,E2 -23983.757} C_VEL
LIN {X 0,Y 219.418,Z 625.089,A -85,B 0,C 180,E1 -23986.593,E2 -23986.593} C_VEL
LIN {X 0,Y 230.104,Z 638.846,A -85,B 0,C 180,E1 -23989.662,E2 -23989.662} C_VEL
LIN {X 0,Y 240.996,Z 650.904,A -85,B 0,C 180,E1 -23992.514,E2 -23992.514} C_VEL
LIN {X 0,Y 251.542,Z 661.441,A -85,B 0,C 180,E1 -23995.156,E2 -23995.156} C_VEL
LIN {X 0,Y 261.364,Z 670.212,A -85,B 0,C 180,E1 -23997.467,E2 -23997.467} C_VEL
LIN {X 0,Y 277.351,Z 682.97,A -85,B 0,C 180,E1 -24000.951,E2 -24000.951} C_VEL
LIN {X 0,Y 287.277,Z 690.387,A -85,B 0,C 180,E1 -24003.007,E2 -24003.007} C_VEL
LIN {X 0,Y 295.12,Z 696.261,A -85,B 0,C 180,E1 -24004.812,E2 -24004.812} C_VEL
LIN {X 0,Y 301.509,Z 700.889,A -85,B 0,C 180,E1 -24006.393,E2 -24006.393} C_VEL
LIN {X 0,Y 308.114,Z 705.678,A -85,B 0,C 180,E1 -24008.176,E2 -24008.176} C_VEL
LIN {X 0,Y 314.227,Z 709.774,A -85,B 0,C 180,E1 -24009.944,E2 -24009.944} C_VEL
LIN {X 0,Y 320.721,Z 714.515,A -85,B 0,C 180,E1 -24012.135,E2 -24012.135} C_VEL
LIN {X 0,Y 325.022,Z 717.333,A -85,B 0,C 180,E1 -24013.674,E2 -24013.674} C_VEL
LIN {X 0,Y 330.152,Z 720.43,A -85,B 0,C 180,E1 -24015.696,E2 -24015.696} C_VEL
LIN {X 0,Y 334.489,Z 723.627,A -85,B 0,C 180,E1 -24017.871,E2 -24017.871} C_VEL
LIN {X 0,Y 336.88,Z 725.21,A -85,B 0,C 180,E1 -24019.178,E2 -24019.178} C_VEL
LIN {X 0,Y 339.009,Z 726.479,A -85,B 0,C 180,E1 -24020.454,E2 -24020.454} C_VEL
LIN {X 0,Y 340.893,Z 727.479,A -85,B 0,C 180,E1 -24021.719,E2 -24021.719} C_VEL
LIN {X 0,Y 342.505,Z 728.256,A -85,B 0,C 180,E1 -24022.928,E2 -24022.928} C_VEL
LIN {X 0,Y 343.856,Z 728.925,A -85,B 0,C 180,E1 -24024.135,E2 -24024.135} C_VEL
LIN {X 0,Y 345.915,Z 729.719,A -85,B 0,C 180,E1 -24026.506,E2 -24026.506} C_VEL
LIN {X 0,Y 346.508,Z 729.988,A -85,B 0,C 180,E1 -24027.675,E2 -24027.675} C_VEL
LIN {X 0,Y 347.046,Z 730.13,A -85,B 0,C 180,E1 -24030,E2 -24030} C_VEL
LIN {X 0,Y 346.511,Z 729.994,A -85,B 0,C 180,E1 -24032.325,E2 -24032.325} C_VEL
LIN {X 0,Y 345.339,Z 729.549,A -85,B 0,C 180,E1 -24034.299,E2 -24034.299} C_VEL
LIN {X 0,Y 343.854,Z 728.921,A -85,B 0,C 180,E1 -24035.865,E2 -24035.865} C_VEL
LIN {X 0,Y 342.493,Z 728.252,A -85,B 0,C 180,E1 -24037.072,E2 -24037.072} C_VEL
LIN {X 0,Y 340.848,Z 727.461,A -85,B 0,C 180,E1 -24038.299,E2 -24038.299} C_VEL
LIN {X 0,Y 338.999,Z 726.449,A -85,B 0,C 180,E1 -24039.547,E2 -24039.547} C_VEL
LIN {X 0,Y 336.531,Z 724.968,A -85,B 0,C 180,E1 -24041.033,E2 -24041.033} C_VEL
LIN {X 0,Y 331.919,Z 721.691,A -85,B 0,C 180,E1 -24043.468,E2 -24043.468} C_VEL
LIN {X 0,Y 327.823,Z 718.961,A -85,B 0,C 180,E1 -24045.266,E2 -24045.266} C_VEL
LIN {X 0,Y 323.293,Z 716.24,A -85,B 0,C 180,E1 -24046.963,E2 -24046.963} C_VEL
LIN {X 0,Y 315.999,Z 711.088,A -85,B 0,C 180,E1 -24049.487,E2 -24049.487} C_VEL
LIN {X 0,Y 309.527,Z 706.646,A -85,B 0,C 180,E1 -24051.422,E2 -24051.422} C_VEL
LIN {X 0,Y 302.971,Z 701.99,A -85,B 0,C 180,E1 -24053.225,E2 -24053.225} C_VEL
LIN {X 0,Y 298.399,Z 698.585,A -85,B 0,C 180,E1 -24054.408,E2 -24054.408} C_VEL
LIN {X 0,Y 290.159,Z 692.604,A -85,B 0,C 180,E1 -24056.341,E2 -24056.341} C_VEL
LIN {X 0,Y 282.268,Z 686.68,A -85,B 0,C 180,E1 -24058.039,E2 -24058.039} C_VEL
LIN {X 0,Y 267.128,Z 675.044,A -85,B 0,C 180,E1 -24061.235,E2 -24061.235} C_VEL
LIN {X 0,Y 254.614,Z 664.363,A -85,B 0,C 180,E1 -24064.1,E2 -24064.1} C_VEL
LIN {X 0,Y 243.614,Z 653.629,A -85,B 0,C 180,E1 -24066.812,E2 -24066.812} C_VEL
LIN {X 0,Y 232.188,Z 641.264,A -85,B 0,C 180,E1 -24069.793,E2 -24069.793} C_VEL
LIN {X 0,Y 221.137,Z 627.466,A -85,B 0,C 180,E1 -24072.881,E2 -24072.881} C_VEL
LIN {X 0,Y 213.684,Z 616.351,A -85,B 0,C 180,E1 -24075.299,E2 -24075.299} C_VEL
LIN {X 0,Y 206.703,Z 603.682,A -85,B 0,C 180,E1 -24077.945,E2 -24077.945} C_VEL
LIN {X 0,Y 199.552,Z 588.379,A -85,B 0,C 180,E1 -24081.147,E2 -24081.147} C_VEL
LIN {X 0,Y 193.914,Z 577.744,A -85,B 0,C 180,E1 -24083.933,E2 -24083.933} C_VEL
LIN {X 0,Y 188.443,Z 568.612,A -85,B 0,C 180,E1 -24086.925,E2 -24086.925} C_VEL
LIN {X 0,Y 183.589,Z 561.249,A -85,B 0,C 180,E1 -24089.91,E2 -24089.91} C_VEL
LIN {X 0,Y 180.86,Z 557.364,A -85,B 0,C 180,E1 -24091.769,E2 -24091.769} C_VEL
LIN {X 0,Y 178.133,Z 553.518,A -85,B 0,C 180,E1 -24093.809,E2 -24093.809} C_VEL
LIN {X 0,Y 174.638,Z 548.869,A -85,B 0,C 180,E1 -24096.742,E2 -24096.742} C_VEL
LIN {X 0,Y 171.854,Z 545.382,A -85,B 0,C 180,E1 -24099.437,E2 -24099.437} C_VEL
LIN {X 0,Y 171.109,Z 544.208,A -85,B 0,C 180,E1 -24100.264,E2 -24100.264} C_VEL
LIN {X 0,Y 168.429,Z 541.427,A -85,B 0,C 180,E1 -24103.428,E2 -24103.428} C_VEL
LIN {X 0,Y 167.162,Z 538.95,A -85,B 0,C 180,E1 -24105.39,E2 -24105.39} C_VEL
LIN {X 0,Y 164.635,Z 537.096,A -85,B 0,C 180,E1 -24109.792,E2 -24109.792} C_VEL
LIN {X 0,Y 162.946,Z 533.879,A -85,B 0,C 180,E1 -24115.672,E2 -24115.672} C_VEL
LIN {X 0,Y 162.627,Z 533.041,A -85,B 0,C 180,E1 -24120.001,E2 -24120.001} C_VEL
LIN {X 0,Y 162.962,Z 533.893,A -85,B 0,C 180,E1 -24124.02,E2 -24124.02} C_VEL
LIN {X 0,Y 166.14,Z 538.427,A -85,B 0,C 180,E1 -24132.677,E2 -24132.677} C_VEL
LIN {X 0,Y 167.341,Z 539.335,A -85,B 0,C 180,E1 -24134.519,E2 -24134.519} C_VEL
LIN {X 0,Y 169.404,Z 542.697,A -85,B 0,C 180,E1 -24137.443,E2 -24137.443} C_VEL
LIN {X 0,Y 171.447,Z 544.638,A -85,B 0,C 180,E1 -24139.711,E2 -24139.711} C_VEL
LIN {X 0,Y 173.895,Z 548.185,A -85,B 0,C 180,E1 -24142.21,E2 -24142.21} C_VEL
LIN {X 0,Y 175.487,Z 549.893,A -85,B 0,C 180,E1 -24143.61,E2 -24143.61} C_VEL
LIN {X 0,Y 179.213,Z 555.027,A -85,B 0,C 180,E1 -24146.63,E2 -24146.63} C_VEL
LIN {X 0,Y 182.595,Z 559.888,A -85,B 0,C 180,E1 -24149.044,E2 -24149.044} C_VEL
LIN {X 0,Y 185.031,Z 563.482,A -85,B 0,C 180,E1 -24150.632,E2 -24150.632} C_VEL
LIN {X 0,Y 189.905,Z 572.9,A -85,B 0,C 180,E1 -24153.645,E2 -24153.645} C_VEL
LIN {X 0,Y 194.982,Z 584.153,A -85,B 0,C 180,E1 -24156.495,E2 -24156.495} C_VEL
LIN {X 0,Y 199.744,Z 596.296,A -85,B 0,C 180,E1 -24158.973,E2 -24158.973} C_VEL
LIN {X 0,Y 200.509,Z 598.494,A -85,B 0,C 180,E1 -24159.361,E2 -24159.361} C_VEL
LIN {X 0,Y 196.778,Z 650.041,A -85,B 0,C 180,E1 -24160.986,E2 -24160.986} C_VEL
LIN {X 0,Y 195.145,Z 662.177,A -85,B 0,C 180,E1 -24161.548,E2 -24161.548} C_VEL
LIN {X 0,Y 193.245,Z 672.253,A -85,B 0,C 180,E1 -24162.184,E2 -24162.184} C_VEL
LIN {X 0,Y 190.908,Z 682.041,A -85,B 0,C 180,E1 -24162.975,E2 -24162.975} C_VEL
LIN {X 0,Y 188.087,Z 692.007,A -85,B 0,C 180,E1 -24164.005,E2 -24164.005} C_VEL
LIN {X 0,Y 184.821,Z 701.923,A -85,B 0,C 180,E1 -24165.294,E2 -24165.294} C_VEL
LIN {X 0,Y 181.099,Z 711.64,A -85,B 0,C 180,E1 -24166.846,E2 -24166.846} C_VEL
LIN {X 0,Y 176.996,Z 721.372,A -85,B 0,C 180,E1 -24168.804,E2 -24168.804} C_VEL
LIN {X 0,Y 172.944,Z 730.076,A -85,B 0,C 180,E1 -24170.96,E2 -24170.96} C_VEL
LIN {X 0,Y 169.419,Z 737.049,A -85,B 0,C 180,E1 -24173.023,E2 -24173.023} C_VEL
LIN {X 0,Y 165.23,Z 744.567,A -85,B 0,C 180,E1 -24175.697,E2 -24175.697} C_VEL
LIN {X 0,Y 160.831,Z 752.177,A -85,B 0,C 180,E1 -24179.107,E2 -24179.107} C_VEL
LIN {X 0,Y 157.61,Z 757.58,A -85,B 0,C 180,E1 -24182.083,E2 -24182.083} C_VEL
LIN {X 0,Y 154.354,Z 763.016,A -85,B 0,C 180,E1 -24185.809,E2 -24185.809} C_VEL
LIN {X 0,Y 151.827,Z 767.468,A -85,B 0,C 180,E1 -24189.686,E2 -24189.686} C_VEL
LIN {X 0,Y 149.784,Z 771.017,A -85,B 0,C 180,E1 -24193.649,E2 -24193.649} C_VEL
LIN {X 0,Y 148.866,Z 772.964,A -85,B 0,C 180,E1 -24196.347,E2 -24196.347} C_VEL
LIN {X 0,Y 147.802,Z 775.665,A -85,B 0,C 180,E1 -24201.799,E2 -24201.799} C_VEL
LIN {X 0,Y 147.611,Z 776.971,A -85,B 0,C 180,E1 -24207.271,E2 -24207.271} C_VEL
LIN {X 0,Y 147.719,Z 777.228,A -85,B 0,C 180,E1 -24210,E2 -24210} C_VEL
LIN {X 0,Y 147.628,Z 776.49,A -85,B 0,C 180,E1 -24215.463,E2 -24215.463} C_VEL
LIN {X 0,Y 147.802,Z 775.665,A -85,B 0,C 180,E1 -24218.201,E2 -24218.201} C_VEL
LIN {X 0,Y 148.866,Z 772.964,A -85,B 0,C 180,E1 -24223.653,E2 -24223.653} C_VEL
LIN {X 0,Y 151.095,Z 768.736,A -85,B 0,C 180,E1 -24229.001,E2 -24229.001} C_VEL
LIN {X 0,Y 153.477,Z 764.598,A -85,B 0,C 180,E1 -24232.906,E2 -24232.906} C_VEL
LIN {X 0,Y 155.598,Z 760.978,A -85,B 0,C 180,E1 -24235.724,E2 -24235.724} C_VEL
LIN {X 0,Y 156.627,Z 758.254,A -85,B 0,C 180,E1 -24237.601,E2 -24237.601} C_VEL
LIN {X 0,Y 157.321,Z 749.038,A -85,B 0,C 180,E1 -24243.587,E2 -24243.587} C_VEL
LIN {X 0,Y 158.36,Z 746.114,A -85,B 0,C 180,E1 -24245.004,E2 -24245.004} C_VEL
LIN {X 0,Y 159.025,Z 744.91,A -85,B 0,C 180,E1 -24245.526,E2 -24245.526} C_VEL
LIN {X 0,Y 164.719,Z 735.281,A -85,B 0,C 180,E1 -24249,E2 -24249} C_VEL
LIN {X 0,Y 170.342,Z 724.196,A -85,B 0,C 180,E1 -24252.041,E2 -24252.041} C_VEL
LIN {X 0,Y 174.437,Z 715.163,A -85,B 0,C 180,E1 -24254.025,E2 -24254.025} C_VEL
LIN {X 0,Y 178.19,Z 706.116,A -85,B 0,C 180,E1 -24255.631,E2 -24255.631} C_VEL
LIN {X 0,Y 182.064,Z 695.314,A -85,B 0,C 180,E1 -24257.174,E2 -24257.174} C_VEL
LIN {X 0,Y 185.271,Z 685.062,A -85,B 0,C 180,E1 -24258.314,E2 -24258.314} C_VEL
LIN {X 0,Y 188.239,Z 673.414,A -85,B 0,C 180,E1 -24259.32,E2 -24259.32} C_VEL
LIN {X 0,Y 190.482,Z 661.978,A -85,B 0,C 180,E1 -24260.061,E2 -24260.061} C_VEL
LIN {X 0,Y 192.081,Z 650.634,A -85,B 0,C 180,E1 -24260.578,E2 -24260.578} C_VEL
LIN {X 0,Y 194.46,Z 621.194,A -85,B 0,C 180,E1 -24261.515,E2 -24261.515} C_VEL
LIN {X 0,Y 195.868,Z 600.748,A -85,B 0,C 180,E1 -24262.18,E2 -24262.18} C_VEL
LIN {X 0,Y 191.349,Z 588.748,A -85,B 0,C 180,E1 -24264.699,E2 -24264.699} C_VEL
LIN {X 0,Y 186.428,Z 577.416,A -85,B 0,C 180,E1 -24267.665,E2 -24267.665} C_VEL
LIN {X 0,Y 181.817,Z 568.252,A -85,B 0,C 180,E1 -24270.733,E2 -24270.733} C_VEL
LIN {X 0,Y 177.489,Z 561.955,A -85,B 0,C 180,E1 -24273.866,E2 -24273.866} C_VEL
LIN {X 0,Y 175.649,Z 559.328,A -85,B 0,C 180,E1 -24275.356,E2 -24275.356} C_VEL
LIN {X 0,Y 172.802,Z 555.38,A -85,B 0,C 180,E1 -24277.9,E2 -24277.9} C_VEL
LIN {X 0,Y 170.079,Z 551.797,A -85,B 0,C 180,E1 -24280.695,E2 -24280.695} C_VEL
LIN {X 0,Y 169.343,Z 550.721,A -85,B 0,C 180,E1 -24281.551,E2 -24281.551} C_VEL
LIN {X 0,Y 166.783,Z 547.7,A -85,B 0,C 180,E1 -24284.836,E2 -24284.836} C_VEL
LIN {X 0,Y 165.764,Z 545.792,A -85,B 0,C 180,E1 -24286.514,E2 -24286.514} C_VEL
LIN {X 0,Y 162.934,Z 543.015,A -85,B 0,C 180,E1 -24292.33,E2 -24292.33} C_VEL
LIN {X 0,Y 161.962,Z 540.643,A -85,B 0,C 180,E1 -24296.89,E2 -24296.89} C_VEL
LIN {X 0,Y 161.766,Z 540.051,A -85,B 0,C 180,E1 -24299.999,E2 -24299.999} C_VEL
LIN {X 0,Y 162.077,Z 541.032,A -85,B 0,C 180,E1 -24304.381,E2 -24304.381} C_VEL
LIN {X 0,Y 164.8,Z 545.22,A -85,B 0,C 180,E1 -24312.31,E2 -24312.31} C_VEL
LIN {X 0,Y 166.033,Z 546.165,A -85,B 0,C 180,E1 -24314.32,E2 -24314.32} C_VEL
LIN {X 0,Y 168.176,Z 549.67,A -85,B 0,C 180,E1 -24317.478,E2 -24317.478} C_VEL
LIN {X 0,Y 169.954,Z 551.488,A -85,B 0,C 180,E1 -24319.539,E2 -24319.539} C_VEL
LIN {X 0,Y 172.725,Z 555.315,A -85,B 0,C 180,E1 -24322.423,E2 -24322.423} C_VEL
LIN {X 0,Y 173.984,Z 556.987,A -85,B 0,C 180,E1 -24323.587,E2 -24323.587} C_VEL
LIN {X 0,Y 177.075,Z 561.37,A -85,B 0,C 180,E1 -24326.201,E2 -24326.201} C_VEL
LIN {X 0,Y 179.971,Z 565.574,A -85,B 0,C 180,E1 -24328.381,E2 -24328.381} C_VEL
LIN {X 0,Y 184.61,Z 572.639,A -85,B 0,C 180,E1 -24331.483,E2 -24331.483} C_VEL
LIN {X 0,Y 189.946,Z 581.738,A -85,B 0,C 180,E1 -24334.639,E2 -24334.639} C_VEL
LIN {X 0,Y 194.744,Z 590.872,A -85,B 0,C 180,E1 -24337.198,E2 -24337.198} C_VEL
LIN {X 0,Y 199.022,Z 600.085,A -85,B 0,C 180,E1 -24339.322,E2 -24339.322} C_VEL
LIN {X 0,Y 206.83,Z 616.308,A -85,B 0,C 180,E1 -24342.733,E2 -24342.733} C_VEL
LIN {X 0,Y 215.161,Z 629.781,A -85,B 0,C 180,E1 -24345.719,E2 -24345.719} C_VEL
LIN {X 0,Y 223.74,Z 641.218,A -85,B 0,C 180,E1 -24348.382,E2 -24348.382} C_VEL
LIN {X 0,Y 231.429,Z 650.432,A -85,B 0,C 180,E1 -24350.614,E2 -24350.614} C_VEL
LIN {X 0,Y 243.371,Z 663.322,A -85,B 0,C 180,E1 -24353.955,E2 -24353.955} C_VEL
LIN {X 0,Y 255.418,Z 674.501,A -85,B 0,C 180,E1 -24357.057,E2 -24357.057} C_VEL
LIN {X 0,Y 270.145,Z 686.272,A -85,B 0,C 180,E1 -24360.483,E2 -24360.483} C_VEL
LIN {X 0,Y 284.199,Z 696.931,A -85,B 0,C 180,E1 -24363.569,E2 -24363.569} C_VEL
LIN {X 0,Y 293.165,Z 703.441,A -85,B 0,C 180,E1 -24365.637,E2 -24365.637} C_VEL
LIN {X 0,Y 299.237,Z 707.93,A -85,B 0,C 180,E1 -24367.212,E2 -24367.212} C_VEL
LIN {X 0,Y 305.17,Z 712.147,A -85,B 0,C 180,E1 -24368.856,E2 -24368.856} C_VEL
LIN {X 0,Y 310.788,Z 715.974,A -85,B 0,C 180,E1 -24370.544,E2 -24370.544} C_VEL
LIN {X 0,Y 314.47,Z 718.677,A -85,B 0,C 180,E1 -24371.767,E2 -24371.767} C_VEL
LIN {X 0,Y 321.326,Z 723.168,A -85,B 0,C 180,E1 -24374.227,E2 -24374.227} C_VEL
LIN {X 0,Y 326.324,Z 726.315,A -85,B 0,C 180,E1 -24376.296,E2 -24376.296} C_VEL
LIN {X 0,Y 330.168,Z 729.103,A -85,B 0,C 180,E1 -24378.279,E2 -24378.279} C_VEL
LIN {X 0,Y 334.552,Z 731.824,A -85,B 0,C 180,E1 -24380.867,E2 -24380.867} C_VEL
LIN {X 0,Y 337.321,Z 733.209,A -85,B 0,C 180,E1 -24382.819,E2 -24382.819} C_VEL
LIN {X 0,Y 339.002,Z 734.04,A -85,B 0,C 180,E1 -24384.323,E2 -24384.323} C_VEL
LIN {X 0,Y 340.883,Z 734.756,A -85,B 0,C 180,E1 -24386.454,E2 -24386.454} C_VEL
LIN {X 0,Y 341.521,Z 735.042,A -85,B 0,C 180,E1 -24387.641,E2 -24387.641} C_VEL
LIN {X 0,Y 342.084,Z 735.212,A -85,B 0,C 180,E1 -24390,E2 -24390} C_VEL
LIN {X 0,Y 341.523,Z 735.05,A -85,B 0,C 180,E1 -24392.359,E2 -24392.359} C_VEL
LIN {X 0,Y 340.889,Z 734.762,A -85,B 0,C 180,E1 -24393.546,E2 -24393.546} C_VEL
LIN {X 0,Y 338.725,Z 733.899,A -85,B 0,C 180,E1 -24395.955,E2 -24395.955} C_VEL
LIN {X 0,Y 337.299,Z 733.215,A -85,B 0,C 180,E1 -24397.182,E2 -24397.182} C_VEL
LIN {X 0,Y 334.561,Z 731.82,A -85,B 0,C 180,E1 -24399.142,E2 -24399.142} C_VEL
LIN {X 0,Y 330.17,Z 729.065,A -85,B 0,C 180,E1 -24401.723,E2 -24401.723} C_VEL
LIN {X 0,Y 325.841,Z 725.938,A -85,B 0,C 180,E1 -24403.932,E2 -24403.932} C_VEL
LIN {X 0,Y 321.325,Z 723.144,A -85,B 0,C 180,E1 -24405.772,E2 -24405.772} C_VEL
LIN {X 0,Y 314.424,Z 718.663,A -85,B 0,C 180,E1 -24408.235,E2 -24408.235} C_VEL
LIN {X 0,Y 309.412,Z 714.906,A -85,B 0,C 180,E1 -24409.92,E2 -24409.92} C_VEL
LIN {X 0,Y 302.79,Z 710.502,A -85,B 0,C 180,E1 -24411.81,E2 -24411.81} C_VEL
LIN {X 0,Y 295.169,Z 704.833,A -85,B 0,C 180,E1 -24413.876,E2 -24413.876} C_VEL
LIN {X 0,Y 288.182,Z 699.893,A -85,B 0,C 180,E1 -24415.536,E2 -24415.536} C_VEL
LIN {X 0,Y 280.587,Z 694.122,A -85,B 0,C 180,E1 -24417.231,E2 -24417.231} C_VEL
LIN {X 0,Y 265.342,Z 682.614,A -85,B 0,C 180,E1 -24420.594,E2 -24420.594} C_VEL
LIN {X 0,Y 250.918,Z 670.555,A -85,B 0,C 180,E1 -24424.068,E2 -24424.068} C_VEL
LIN {X 0,Y 239.403,Z 659.15,A -85,B 0,C 180,E1 -24427.137,E2 -24427.137} C_VEL
LIN {X 0,Y 227.405,Z 645.772,A -85,B 0,C 180,E1 -24430.556,E2 -24430.556} C_VEL
LIN {X 0,Y 217.169,Z 632.594,A -85,B 0,C 180,E1 -24433.637,E2 -24433.637} C_VEL
LIN {X 0,Y 209.402,Z 620.738,A -85,B 0,C 180,E1 -24436.289,E2 -24436.289} C_VEL
LIN {X 0,Y 202.607,Z 608.025,A -85,B 0,C 180,E1 -24439.024,E2 -24439.024} C_VEL
LIN {X 0,Y 195.723,Z 592.823,A -85,B 0,C 180,E1 -24442.307,E2 -24442.307} C_VEL
LIN {X 0,Y 190.621,Z 582.949,A -85,B 0,C 180,E1 -24444.988,E2 -24444.988} C_VEL
LIN {X 0,Y 185.393,Z 573.939,A -85,B 0,C 180,E1 -24448.027,E2 -24448.027} C_VEL
LIN {X 0,Y 180.805,Z 566.847,A -85,B 0,C 180,E1 -24451.027,E2 -24451.027} C_VEL
LIN {X 0,Y 178.083,Z 562.859,A -85,B 0,C 180,E1 -24453.011,E2 -24453.011} C_VEL
LIN {X 0,Y 175.865,Z 559.621,A -85,B 0,C 180,E1 -24454.784,E2 -24454.784} C_VEL
LIN {X 0,Y 172.876,Z 555.451,A -85,B 0,C 180,E1 -24457.44,E2 -24457.44} C_VEL
LIN {X 0,Y 169.995,Z 551.591,A -85,B 0,C 180,E1 -24460.409,E2 -24460.409} C_VEL
LIN {X 0,Y 169.019,Z 550.5,A -85,B 0,C 180,E1 -24461.516,E2 -24461.516} C_VEL
LIN {X 0,Y 166.516,Z 547.206,A -85,B 0,C 180,E1 -24464.863,E2 -24464.863} C_VEL
LIN {X 0,Y 165.909,Z 545.868,A -85,B 0,C 180,E1 -24465.904,E2 -24465.904} C_VEL
LIN {X 0,Y 163.246,Z 543.569,A -85,B 0,C 180,E1 -24471.023,E2 -24471.023} C_VEL
LIN {X 0,Y 161.995,Z 540.777,A -85,B 0,C 180,E1 -24476.206,E2 -24476.206} C_VEL
LIN {X 0,Y 161.761,Z 540.092,A -85,B 0,C 180,E1 -24480.001,E2 -24480.001} C_VEL
LIN {X 0,Y 162.091,Z 541.001,A -85,B 0,C 180,E1 -24484.041,E2 -24484.041} C_VEL
LIN {X 0,Y 165.023,Z 545.333,A -85,B 0,C 180,E1 -24492.296,E2 -24492.296} C_VEL
LIN {X 0,Y 165.988,Z 546.121,A -85,B 0,C 180,E1 -24493.857,E2 -24493.857} C_VEL
LIN {X 0,Y 168.344,Z 549.817,A -85,B 0,C 180,E1 -24497.289,E2 -24497.289} C_VEL
LIN {X 0,Y 169.842,Z 551.328,A -85,B 0,C 180,E1 -24499.019,E2 -24499.019} C_VEL
LIN {X 0,Y 172.357,Z 554.935,A -85,B 0,C 180,E1 -24501.688,E2 -24501.688} C_VEL
LIN {X 0,Y 173.619,Z 556.394,A -85,B 0,C 180,E1 -24502.853,E2 -24502.853} C_VEL
LIN {X 0,Y 177.159,Z 561.475,A -85,B 0,C 180,E1 -24505.874,E2 -24505.874} C_VEL
LIN {X 0,Y 181.01,Z 567.113,A -85,B 0,C 180,E1 -24508.72,E2 -24508.72} C_VEL
LIN {X 0,Y 182.936,Z 570.352,A -85,B 0,C 180,E1 -24510.043,E2 -24510.043} C_VEL
LIN {X 0,Y 187.458,Z 579.765,A -85,B 0,C 180,E1 -24512.987,E2 -24512.987} C_VEL
LIN {X 0,Y 191.519,Z 589.173,A -85,B 0,C 180,E1 -24515.399,E2 -24515.399} C_VEL
LIN {X 0,Y 195.759,Z 600.41,A -85,B 0,C 180,E1 -24517.759,E2 -24517.759} C_VEL
LIN {X 0,Y 195.795,Z 603.17,A -85,B 0,C 180,E1 -24517.934,E2 -24517.934} C_VEL
LIN {X 0,Y 192.1,Z 650.81,A -85,B 0,C 180,E1 -24519.429,E2 -24519.429} C_VEL
LIN {X 0,Y 190.206,Z 663.803,A -85,B 0,C 180,E1 -24520.046,E2 -24520.046} C_VEL
LIN {X 0,Y 187.048,Z 678.625,A -85,B 0,C 180,E1 -24521.08,E2 -24521.08} C_VEL
LIN {X 0,Y 183.799,Z 690.056,A -85,B 0,C 180,E1 -24522.198,E2 -24522.198} C_VEL
LIN {X 0,Y 179.848,Z 701.725,A -85,B 0,C 180,E1 -24523.704,E2 -24523.704} C_VEL
LIN {X 0,Y 175.981,Z 711.442,A -85,B 0,C 180,E1 -24525.263,E2 -24525.263} C_VEL
LIN {X 0,Y 171.858,Z 720.862,A -85,B 0,C 180,E1 -24527.169,E2 -24527.169} C_VEL
LIN {X 0,Y 167.468,Z 729.877,A -85,B 0,C 180,E1 -24529.424,E2 -24529.424} C_VEL
LIN {X 0,Y 163.789,Z 736.85,A -85,B 0,C 180,E1 -24531.526,E2 -24531.526} C_VEL
LIN {X 0,Y 159.367,Z 744.367,A -85,B 0,C 180,E1 -24534.246,E2 -24534.246} C_VEL
LIN {X 0,Y 154.747,Z 751.978,A -85,B 0,C 180,E1 -24537.749,E2 -24537.749} C_VEL
LIN {X 0,Y 151.334,Z 757.381,A -85,B 0,C 180,E1 -24540.816,E2 -24540.816} C_VEL
LIN {X 0,Y 147.855,Z 762.816,A -85,B 0,C 180,E1 -24544.673,E2 -24544.673} C_VEL
LIN {X 0,Y 145.122,Z 767.268,A -85,B 0,C 180,E1 -24548.703,E2 -24548.703} C_VEL
LIN {X 0,Y 142.949,Z 770.818,A -85,B 0,C 180,E1 -24552.844,E2 -24552.844} C_VEL
LIN {X 0,Y 141.935,Z 772.765,A -85,B 0,C 180,E1 -24555.666,E2 -24555.666} C_VEL
LIN {X 0,Y 140.762,Z 775.466,A -85,B 0,C 180,E1 -24561.386,E2 -24561.386} C_VEL
LIN {X 0,Y 140.508,Z 776.773,A -85,B 0,C 180,E1 -24567.133,E2 -24567.133} C_VEL
LIN {X 0,Y 140.572,Z 776.987,A -85,B 0,C 180,E1 -24570.644,E2 -24570.644} C_VEL
LIN {X 0,Y 140.545,Z 776.292,A -85,B 0,C 180,E1 -24575.74,E2 -24575.74} C_VEL
LIN {X 0,Y 140.762,Z 775.466,A -85,B 0,C 180,E1 -24578.614,E2 -24578.614} C_VEL
LIN {X 0,Y 141.935,Z 772.765,A -85,B 0,C 180,E1 -24584.334,E2 -24584.334} C_VEL
LIN {X 0,Y 144.362,Z 768.537,A -85,B 0,C 180,E1 -24589.924,E2 -24589.924} C_VEL
LIN {X 0,Y 146.888,Z 764.398,A -85,B 0,C 180,E1 -24593.997,E2 -24593.997} C_VEL
LIN {X 0,Y 150.109,Z 759.295,A -85,B 0,C 180,E1 -24597.916,E2 -24597.916} C_VEL
LIN {X 0,Y 154.014,Z 753.115,A -85,B 0,C 180,E1 -24601.652,E2 -24601.652} C_VEL
LIN {X 0,Y 157.733,Z 747.041,A -85,B 0,C 180,E1 -24604.616,E2 -24604.616} C_VEL
LIN {X 0,Y 159.025,Z 744.91,A -85,B 0,C 180,E1 -24605.526,E2 -24605.526} C_VEL
LIN {X 0,Y 160.688,Z 741.328,A -85,B 0,C 180,E1 -24607.102,E2 -24607.102} C_VEL
LIN {X 0,Y 161.97,Z 735.196,A -85,B 0,C 180,E1 -24609.844,E2 -24609.844} C_VEL
LIN {X 0,Y 163.327,Z 728.572,A -85,B 0,C 180,E1 -24612.403,E2 -24612.403} C_VEL
LIN {X 0,Y 165.03,Z 724.186,A -85,B 0,C 180,E1 -24613.651,E2 -24613.651} C_VEL
LIN {X 0,Y 169.393,Z 714.964,A -85,B 0,C 180,E1 -24615.698,E2 -24615.698} C_VEL
LIN {X 0,Y 173.294,Z 705.917,A -85,B 0,C 180,E1 -24617.311,E2 -24617.311} C_VEL
LIN {X 0,Y 177.304,Z 695.116,A -85,B 0,C 180,E1 -24618.86,E2 -24618.86} C_VEL
LIN {X 0,Y 180.637,Z 684.865,A -85,B 0,C 180,E1 -24619.992,E2 -24619.992} C_VEL
LIN {X 0,Y 183.698,Z 673.216,A -85,B 0,C 180,E1 -24620.996,E2 -24620.996} C_VEL
LIN {X 0,Y 186.01,Z 661.781,A -85,B 0,C 180,E1 -24621.735,E2 -24621.735} C_VEL
LIN {X 0,Y 187.649,Z 650.575,A -85,B 0,C 180,E1 -24622.242,E2 -24622.242} C_VEL
LIN {X 0,Y 190.256,Z 619.266,A -85,B 0,C 180,E1 -24623.243,E2 -24623.243} C_VEL
LIN {X 0,Y 191.428,Z 603.219,A -85,B 0,C 180,E1 -24623.761,E2 -24623.761} C_VEL
LIN {X 0,Y 186.96,Z 591.115,A -85,B 0,C 180,E1 -24626.47,E2 -24626.47} C_VEL
LIN {X 0,Y 181.956,Z 579.58,A -85,B 0,C 180,E1 -24629.779,E2 -24629.779} C_VEL
LIN {X 0,Y 178.937,Z 573.593,A -85,B 0,C 180,E1 -24631.962,E2 -24631.962} C_VEL
LIN {X 0,Y 174.027,Z 566.092,A -85,B 0,C 180,E1 -24635.864,E2 -24635.864} C_VEL
LIN {X 0,Y 170.926,Z 561.784,A -85,B 0,C 180,E1 -24638.755,E2 -24638.755} C_VEL
LIN {X 0,Y 168.225,Z 557.918,A -85,B 0,C 180,E1 -24641.739,E2 -24641.739} C_VEL
LIN {X 0,Y 165.208,Z 554.029,A -85,B 0,C 180,E1 -24645.84,E2 -24645.84} C_VEL
LIN {X 0,Y 164.535,Z 552.663,A -85,B 0,C 180,E1 -24647.04,E2 -24647.04} C_VEL
LIN {X 0,Y 161.806,Z 549.7,A -85,B 0,C 180,E1 -24653.139,E2 -24653.139} C_VEL
LIN {X 0,Y 161.024,Z 547.542,A -85,B 0,C 180,E1 -24657.497,E2 -24657.497} C_VEL
LIN {X 0,Y 160.903,Z 547.083,A -85,B 0,C 180,E1 -24659.999,E2 -24659.999} C_VEL
LIN {X 0,Y 161.198,Z 548.154,A -85,B 0,C 180,E1 -24664.375,E2 -24664.375} C_VEL
LIN {X 0,Y 163.705,Z 552.165,A -85,B 0,C 180,E1 -24671.941,E2 -24671.941} C_VEL
LIN {X 0,Y 164.744,Z 553.021,A -85,B 0,C 180,E1 -24673.726,E2 -24673.726} C_VEL
LIN {X 0,Y 167.086,Z 556.755,A -85,B 0,C 180,E1 -24677.28,E2 -24677.28} C_VEL
LIN {X 0,Y 168.4,Z 558.212,A -85,B 0,C 180,E1 -24678.87,E2 -24678.87} C_VEL
LIN {X 0,Y 171.233,Z 562.098,A -85,B 0,C 180,E1 -24681.933,E2 -24681.933} C_VEL
LIN {X 0,Y 175.09,Z 567.805,A -85,B 0,C 180,E1 -24685.449,E2 -24685.449} C_VEL
LIN {X 0,Y 179.331,Z 574.185,A -85,B 0,C 180,E1 -24688.713,E2 -24688.713} C_VEL
LIN {X 0,Y 184.568,Z 582.986,A -85,B 0,C 180,E1 -24692.213,E2 -24692.213} C_VEL
LIN {X 0,Y 189.562,Z 592.387,A -85,B 0,C 180,E1 -24695.165,E2 -24695.165} C_VEL
LIN {X 0,Y 194.323,Z 602.51,A -85,B 0,C 180,E1 -24697.73,E2 -24697.73} C_VEL
LIN {X 0,Y 201.999,Z 619.354,A -85,B 0,C 180,E1 -24701.379,E2 -24701.379} C_VEL
LIN {X 0,Y 210.808,Z 634.25,A -85,B 0,C 180,E1 -24704.758,E2 -24704.758} C_VEL
LIN {X 0,Y 219.931,Z 646.792,A -85,B 0,C 180,E1 -24707.807,E2 -24707.807} C_VEL
LIN {X 0,Y 228.86,Z 657.752,A -85,B 0,C 180,E1 -24710.666,E2 -24710.666} C_VEL
LIN {X 0,Y 241.101,Z 670.883,A -85,B 0,C 180,E1 -24714.34,E2 -24714.34} C_VEL
LIN {X 0,Y 252.358,Z 681.171,A -85,B 0,C 180,E1 -24717.397,E2 -24717.397} C_VEL
LIN {X 0,Y 268.371,Z 693.825,A -85,B 0,C 180,E1 -24721.315,E2 -24721.315} C_VEL
LIN {X 0,Y 281.03,Z 703.196,A -85,B 0,C 180,E1 -24724.194,E2 -24724.194} C_VEL
LIN {X 0,Y 288.553,Z 708.619,A -85,B 0,C 180,E1 -24725.97,E2 -24725.97} C_VEL
LIN {X 0,Y 294.776,Z 713.244,A -85,B 0,C 180,E1 -24727.576,E2 -24727.576} C_VEL
LIN {X 0,Y 301.997,Z 718.247,A -85,B 0,C 180,E1 -24729.57,E2 -24729.57} C_VEL
LIN {X 0,Y 307.621,Z 722.273,A -85,B 0,C 180,E1 -24731.347,E2 -24731.347} C_VEL
LIN {X 0,Y 314.655,Z 727.028,A -85,B 0,C 180,E1 -24733.825,E2 -24733.825} C_VEL
LIN {X 0,Y 320.261,Z 730.489,A -85,B 0,C 180,E1 -24736.032,E2 -24736.032} C_VEL
LIN {X 0,Y 323.664,Z 732.982,A -85,B 0,C 180,E1 -24737.717,E2 -24737.717} C_VEL
LIN {X 0,Y 328.073,Z 735.853,A -85,B 0,C 180,E1 -24740.198,E2 -24740.198} C_VEL
LIN {X 0,Y 330.029,Z 736.932,A -85,B 0,C 180,E1 -24741.427,E2 -24741.427} C_VEL
LIN {X 0,Y 332.565,Z 738.211,A -85,B 0,C 180,E1 -24743.326,E2 -24743.326} C_VEL
LIN {X 0,Y 334.461,Z 739.118,A -85,B 0,C 180,E1 -24745.179,E2 -24745.179} C_VEL
LIN {X 0,Y 335.499,Z 739.465,A -85,B 0,C 180,E1 -24746.397,E2 -24746.397} C_VEL
LIN {X 0,Y 336.198,Z 739.744,A -85,B 0,C 180,E1 -24747.604,E2 -24747.604} C_VEL
LIN {X 0,Y 336.806,Z 739.928,A -85,B 0,C 180,E1 -24750,E2 -24750} C_VEL
LIN {X 0,Y 336.199,Z 739.751,A -85,B 0,C 180,E1 -24752.396,E2 -24752.396} C_VEL
LIN {X 0,Y 335.507,Z 739.468,A -85,B 0,C 180,E1 -24753.603,E2 -24753.603} C_VEL
LIN {X 0,Y 333.263,Z 738.544,A -85,B 0,C 180,E1 -24756.053,E2 -24756.053} C_VEL
LIN {X 0,Y 331.77,Z 737.834,A -85,B 0,C 180,E1 -24757.302,E2 -24757.302} C_VEL
LIN {X 0,Y 330.016,Z 736.915,A -85,B 0,C 180,E1 -24758.573,E2 -24758.573} C_VEL
LIN {X 0,Y 327.961,Z 735.755,A -85,B 0,C 180,E1 -24759.871,E2 -24759.871} C_VEL
LIN {X 0,Y 323.69,Z 732.931,A -85,B 0,C 180,E1 -24762.304,E2 -24762.304} C_VEL
LIN {X 0,Y 319.264,Z 729.82,A -85,B 0,C 180,E1 -24764.405,E2 -24764.405} C_VEL
LIN {X 0,Y 314.661,Z 727.03,A -85,B 0,C 180,E1 -24766.179,E2 -24766.179} C_VEL
LIN {X 0,Y 310.043,Z 724.004,A -85,B 0,C 180,E1 -24767.818,E2 -24767.818} C_VEL
LIN {X 0,Y 305.45,Z 720.575,A -85,B 0,C 180,E1 -24769.38,E2 -24769.38} C_VEL
LIN {X 0,Y 298.955,Z 716.194,A -85,B 0,C 180,E1 -24771.296,E2 -24771.296} C_VEL
LIN {X 0,Y 291.042,Z 710.427,A -85,B 0,C 180,E1 -24773.423,E2 -24773.423} C_VEL
LIN {X 0,Y 283.541,Z 705.063,A -85,B 0,C 180,E1 -24775.216,E2 -24775.216} C_VEL
LIN {X 0,Y 273.177,Z 697.373,A -85,B 0,C 180,E1 -24777.586,E2 -24777.586} C_VEL
LIN {X 0,Y 257.925,Z 685.813,A -85,B 0,C 180,E1 -24781.178,E2 -24781.178} C_VEL
LIN {X 0,Y 245.193,Z 674.808,A -85,B 0,C 180,E1 -24784.508,E2 -24784.508} C_VEL
LIN {X 0,Y 235.924,Z 665.591,A -85,B 0,C 180,E1 -24787.17,E2 -24787.17} C_VEL
LIN {X 0,Y 224.801,Z 653.011,A -85,B 0,C 180,E1 -24790.596,E2 -24790.596} C_VEL
LIN {X 0,Y 215.119,Z 640.451,A -85,B 0,C 180,E1 -24793.772,E2 -24793.772} C_VEL
LIN {X 0,Y 206.361,Z 627.174,A -85,B 0,C 180,E1 -24796.863,E2 -24796.863} C_VEL
LIN {X 0,Y 199.217,Z 613.703,A -85,B 0,C 180,E1 -24799.854,E2 -24799.854} C_VEL
LIN {X 0,Y 191.978,Z 597.297,A -85,B 0,C 180,E1 -24803.512,E2 -24803.512} C_VEL
LIN {X 0,Y 186.696,Z 586.775,A -85,B 0,C 180,E1 -24806.496,E2 -24806.496} C_VEL
LIN {X 0,Y 181.229,Z 577.285,A -85,B 0,C 180,E1 -24809.959,E2 -24809.959} C_VEL
LIN {X 0,Y 176.524,Z 569.906,A -85,B 0,C 180,E1 -24813.392,E2 -24813.392} C_VEL
LIN {X 0,Y 173.583,Z 565.611,A -85,B 0,C 180,E1 -24815.845,E2 -24815.845} C_VEL
LIN {X 0,Y 170.998,Z 561.868,A -85,B 0,C 180,E1 -24818.292,E2 -24818.292} C_VEL
LIN {X 0,Y 167.801,Z 557.43,A -85,B 0,C 180,E1 -24821.851,E2 -24821.851} C_VEL
LIN {X 0,Y 165.252,Z 554.104,A -85,B 0,C 180,E1 -24825.375,E2 -24825.375} C_VEL
LIN {X 0,Y 164.482,Z 552.674,A -85,B 0,C 180,E1 -24826.724,E2 -24826.724} C_VEL
LIN {X 0,Y 162.057,Z 550.214,A -85,B 0,C 180,E1 -24831.899,E2 -24831.899} C_VEL
LIN {X 0,Y 161.115,Z 547.867,A -85,B 0,C 180,E1 -24836.25,E2 -24836.25} C_VEL
LIN {X 0,Y 160.898,Z 547.12,A -85,B 0,C 180,E1 -24840.001,E2 -24840.001} C_VEL
LIN {X 0,Y 161.174,Z 547.982,A -85,B 0,C 180,E1 -24843.751,E2 -24843.751} C_VEL
LIN {X 0,Y 163.826,Z 552.202,A -85,B 0,C 180,E1 -24851.759,E2 -24851.759} C_VEL
LIN {X 0,Y 164.701,Z 552.963,A -85,B 0,C 180,E1 -24853.26,E2 -24853.26} C_VEL
LIN {X 0,Y 167.148,Z 556.786,A -85,B 0,C 180,E1 -24856.961,E2 -24856.961} C_VEL
LIN {X 0,Y 168.342,Z 558.11,A -85,B 0,C 180,E1 -24858.406,E2 -24858.406} C_VEL
LIN {X 0,Y 170.783,Z 561.634,A -85,B 0,C 180,E1 -24861.106,E2 -24861.106} C_VEL
LIN {X 0,Y 172.134,Z 563.481,A -85,B 0,C 180,E1 -24862.427,E2 -24862.427} C_VEL
LIN {X 0,Y 175.04,Z 567.727,A -85,B 0,C 180,E1 -24865.015,E2 -24865.015} C_VEL
LIN {X 0,Y 179.294,Z 574.181,A -85,B 0,C 180,E1 -24868.299,E2 -24868.299} C_VEL
LIN {X 0,Y 183.423,Z 582.795,A -85,B 0,C 180,E1 -24871.23,E2 -24871.23} C_VEL
LIN {X 0,Y 187.91,Z 593.604,A -85,B 0,C 180,E1 -24874.127,E2 -24874.127} C_VEL
LIN {X 0,Y 191.425,Z 603.245,A -85,B 0,C 180,E1 -24876.24,E2 -24876.24} C_VEL
LIN {X 0,Y 187.661,Z 650.747,A -85,B 0,C 180,E1 -24877.762,E2 -24877.762} C_VEL
LIN {X 0,Y 185.727,Z 663.605,A -85,B 0,C 180,E1 -24878.373,E2 -24878.373} C_VEL
LIN {X 0,Y 182.468,Z 678.427,A -85,B 0,C 180,E1 -24879.401,E2 -24879.401} C_VEL
LIN {X 0,Y 179.098,Z 689.857,A -85,B 0,C 180,E1 -24880.511,E2 -24880.511} C_VEL
LIN {X 0,Y 175.011,Z 701.526,A -85,B 0,C 180,E1 -24882.021,E2 -24882.021} C_VEL
LIN {X 0,Y 170.995,Z 711.243,A -85,B 0,C 180,E1 -24883.583,E2 -24883.583} C_VEL
LIN {X 0,Y 166.541,Z 720.977,A -85,B 0,C 180,E1 -24885.575,E2 -24885.575} C_VEL
LIN {X 0,Y 162.648,Z 728.732,A -85,B 0,C 180,E1 -24887.518,E2 -24887.518} C_VEL
LIN {X 0,Y 158.265,Z 736.651,A -85,B 0,C 180,E1 -24889.918,E2 -24889.918} C_VEL
LIN {X 0,Y 153.634,Z 744.168,A -85,B 0,C 180,E1 -24892.692,E2 -24892.692} C_VEL
LIN {X 0,Y 148.749,Z 751.779,A -85,B 0,C 180,E1 -24896.279,E2 -24896.279} C_VEL
LIN {X 0,Y 145.13,Z 757.181,A -85,B 0,C 180,E1 -24899.439,E2 -24899.439} C_VEL
LIN {X 0,Y 141.438,Z 762.617,A -85,B 0,C 180,E1 -24903.436,E2 -24903.436} C_VEL
LIN {X 0,Y 138.472,Z 767.068,A -85,B 0,C 180,E1 -24907.626,E2 -24907.626} C_VEL
LIN {X 0,Y 136.151,Z 770.619,A -85,B 0,C 180,E1 -24911.958,E2 -24911.958} C_VEL
LIN {X 0,Y 135.009,Z 772.565,A -85,B 0,C 180,E1 -24914.914,E2 -24914.914} C_VEL
LIN {X 0,Y 133.714,Z 775.267,A -85,B 0,C 180,E1 -24920.928,E2 -24920.928} C_VEL
LIN {X 0,Y 133.409,Z 776.574,A -85,B 0,C 180,E1 -24926.98,E2 -24926.98} C_VEL
LIN {X 0,Y 133.535,Z 776.833,A -85,B 0,C 180,E1 -24930,E2 -24930} C_VEL
LIN {X 0,Y 133.457,Z 776.093,A -85,B 0,C 180,E1 -24936.046,E2 -24936.046} C_VEL
LIN {X 0,Y 133.714,Z 775.267,A -85,B 0,C 180,E1 -24939.072,E2 -24939.072} C_VEL
LIN {X 0,Y 135.008,Z 772.565,A -85,B 0,C 180,E1 -24945.086,E2 -24945.086} C_VEL
LIN {X 0,Y 137.651,Z 768.337,A -85,B 0,C 180,E1 -24950.94,E2 -24950.94} C_VEL
LIN {X 0,Y 140.337,Z 764.25,A -85,B 0,C 180,E1 -24955.14,E2 -24955.14} C_VEL
LIN {X 0,Y 143.814,Z 759.095,A -85,B 0,C 180,E1 -24959.253,E2 -24959.253} C_VEL
LIN {X 0,Y 147.986,Z 752.916,A -85,B 0,C 180,E1 -24963.102,E2 -24963.102} C_VEL
LIN {X 0,Y 151.908,Z 746.842,A -85,B 0,C 180,E1 -24966.147,E2 -24966.147} C_VEL
LIN {X 0,Y 156.369,Z 739.773,A -85,B 0,C 180,E1 -24968.992,E2 -24968.992} C_VEL
LIN {X 0,Y 160.172,Z 733.315,A -85,B 0,C 180,E1 -24971.159,E2 -24971.159} C_VEL
LIN {X 0,Y 165.03,Z 724.186,A -85,B 0,C 180,E1 -24973.651,E2 -24973.651} C_VEL
LIN {X 0,Y 166.701,Z 719.841,A -85,B 0,C 180,E1 -24974.838,E2 -24974.838} C_VEL
LIN {X 0,Y 169.033,Z 706.293,A -85,B 0,C 180,E1 -24978.733,E2 -24978.733} C_VEL
LIN {X 0,Y 170.363,Z 701.298,A -85,B 0,C 180,E1 -24979.762,E2 -24979.762} C_VEL
LIN {X 0,Y 171.002,Z 699.582,A -85,B 0,C 180,E1 -24980.033,E2 -24980.033} C_VEL
LIN {X 0,Y 175.848,Z 685.74,A -85,B 0,C 180,E1 -24981.658,E2 -24981.658} C_VEL
LIN {X 0,Y 178.989,Z 674.377,A -85,B 0,C 180,E1 -24982.664,E2 -24982.664} C_VEL
LIN {X 0,Y 181.551,Z 662.495,A -85,B 0,C 180,E1 -24983.44,E2 -24983.44} C_VEL
LIN {X 0,Y 183.326,Z 650.897,A -85,B 0,C 180,E1 -24983.979,E2 -24983.979} C_VEL
LIN {X 0,Y 185.628,Z 624.812,A -85,B 0,C 180,E1 -24984.821,E2 -24984.821} C_VEL
LIN {X 0,Y 187.107,Z 605.66,A -85,B 0,C 180,E1 -24985.432,E2 -24985.432} C_VEL
LIN {X 0,Y 182.834,Z 593.923,A -85,B 0,C 180,E1 -24988.254,E2 -24988.254} C_VEL
LIN {X 0,Y 178.57,Z 583.823,A -85,B 0,C 180,E1 -24991.335,E2 -24991.335} C_VEL
LIN {X 0,Y 176.152,Z 578.989,A -85,B 0,C 180,E1 -24993.219,E2 -24993.219} C_VEL
LIN {X 0,Y 171.763,Z 572.038,A -85,B 0,C 180,E1 -24996.966,E2 -24996.966} C_VEL
LIN {X 0,Y 169.125,Z 568.208,A -85,B 0,C 180,E1 -24999.593,E2 -24999.593} C_VEL
LIN {X 0,Y 166.178,Z 563.942,A -85,B 0,C 180,E1 -25003.096,E2 -25003.096} C_VEL
LIN {X 0,Y 163.69,Z 560.361,A -85,B 0,C 180,E1 -25006.854,E2 -25006.854} C_VEL
LIN {X 0,Y 163.14,Z 559.451,A -85,B 0,C 180,E1 -25007.876,E2 -25007.876} C_VEL
LIN {X 0,Y 160.496,Z 555.81,A -85,B 0,C 180,E1 -25014.975,E2 -25014.975} C_VEL
LIN {X 0,Y 160.064,Z 554.325,A -85,B 0,C 180,E1 -25018.741,E2 -25018.741} C_VEL
LIN {X 0,Y 160.041,Z 554.319,A -85,B 0,C 180,E1 -25021.257,E2 -25021.257} C_VEL
LIN {X 0,Y 160.386,Z 555.483,A -85,B 0,C 180,E1 -25024.79,E2 -25024.79} C_VEL
LIN {X 0,Y 162.617,Z 559.107,A -85,B 0,C 180,E1 -25031.567,E2 -25031.567} C_VEL
LIN {X 0,Y 163.515,Z 559.94,A -85,B 0,C 180,E1 -25033.198,E2 -25033.198} C_VEL
LIN {X 0,Y 165.888,Z 563.702,A -85,B 0,C 180,E1 -25036.932,E2 -25036.932} C_VEL
LIN {X 0,Y 166.808,Z 564.776,A -85,B 0,C 180,E1 -25038.102,E2 -25038.102} C_VEL
LIN {X 0,Y 170.223,Z 569.81,A -85,B 0,C 180,E1 -25041.941,E2 -25041.941} C_VEL
LIN {X 0,Y 173.154,Z 574.303,A -85,B 0,C 180,E1 -25044.699,E2 -25044.699} C_VEL
LIN {X 0,Y 176.921,Z 580.19,A -85,B 0,C 180,E1 -25047.762,E2 -25047.762} C_VEL
LIN {X 0,Y 182.079,Z 589.184,A -85,B 0,C 180,E1 -25051.403,E2 -25051.403} C_VEL
LIN {X 0,Y 186.908,Z 598.776,A -85,B 0,C 180,E1 -25054.414,E2 -25054.414} C_VEL
LIN {X 0,Y 191.184,Z 608.422,A -85,B 0,C 180,E1 -25056.854,E2 -25056.854} C_VEL
LIN {X 0,Y 198.218,Z 624.255,A -85,B 0,C 180,E1 -25060.384,E2 -25060.384} C_VEL
LIN {X 0,Y 206.773,Z 639.164,A -85,B 0,C 180,E1 -25063.881,E2 -25063.881} C_VEL
LIN {X 0,Y 214.803,Z 650.78,A -85,B 0,C 180,E1 -25066.849,E2 -25066.849} C_VEL
LIN {X 0,Y 223.124,Z 661.47,A -85,B 0,C 180,E1 -25069.801,E2 -25069.801} C_VEL
LIN {X 0,Y 234.074,Z 673.83,A -85,B 0,C 180,E1 -25073.431,E2 -25073.431} C_VEL
LIN {X 0,Y 245.811,Z 684.934,A -85,B 0,C 180,E1 -25076.916,E2 -25076.916} C_VEL
LIN {X 0,Y 258.797,Z 695.338,A -85,B 0,C 180,E1 -25080.341,E2 -25080.341} C_VEL
LIN {X 0,Y 273.754,Z 706.329,A -85,B 0,C 180,E1 -25083.965,E2 -25083.965} C_VEL
LIN {X 0,Y 283.868,Z 713.631,A -85,B 0,C 180,E1 -25086.352,E2 -25086.352} C_VEL
LIN {X 0,Y 290.787,Z 718.746,A -85,B 0,C 180,E1 -25088.161,E2 -25088.161} C_VEL
LIN {X 0,Y 296.101,Z 722.419,A -85,B 0,C 180,E1 -25089.64,E2 -25089.64} C_VEL
LIN {X 0,Y 301.658,Z 726.325,A -85,B 0,C 180,E1 -25091.359,E2 -25091.359} C_VEL
LIN {X 0,Y 307.843,Z 730.621,A -85,B 0,C 180,E1 -25093.504,E2 -25093.504} C_VEL
LIN {X 0,Y 313.738,Z 734.262,A -85,B 0,C 180,E1 -25095.735,E2 -25095.735} C_VEL
LIN {X 0,Y 317.01,Z 736.552,A -85,B 0,C 180,E1 -25097.278,E2 -25097.278} C_VEL
LIN {X 0,Y 319.522,Z 738.314,A -85,B 0,C 180,E1 -25098.583,E2 -25098.583} C_VEL
LIN {X 0,Y 321.896,Z 739.855,A -85,B 0,C 180,E1 -25099.941,E2 -25099.941} C_VEL
LIN {X 0,Y 324.052,Z 741.086,A -85,B 0,C 180,E1 -25101.268,E2 -25101.268} C_VEL
LIN {X 0,Y 325.99,Z 742.1,A -85,B 0,C 180,E1 -25102.611,E2 -25102.611} C_VEL
LIN {X 0,Y 327.502,Z 742.833,A -85,B 0,C 180,E1 -25103.841,E2 -25103.841} C_VEL
LIN {X 0,Y 329.823,Z 743.818,A -85,B 0,C 180,E1 -25106.335,E2 -25106.335} C_VEL
LIN {X 0,Y 330.602,Z 744.097,A -85,B 0,C 180,E1 -25107.597,E2 -25107.597} C_VEL
LIN {X 0,Y 331.226,Z 744.29,A -85,B 0,C 180,E1 -25110,E2 -25110} C_VEL
LIN {X 0,Y 330.564,Z 744.114,A -85,B 0,C 180,E1 -25112.437,E2 -25112.437} C_VEL
LIN {X 0,Y 329.828,Z 743.823,A -85,B 0,C 180,E1 -25113.665,E2 -25113.665} C_VEL
LIN {X 0,Y 328.769,Z 743.423,A -85,B 0,C 180,E1 -25114.905,E2 -25114.905} C_VEL
LIN {X 0,Y 327.5,Z 742.826,A -85,B 0,C 180,E1 -25116.159,E2 -25116.159} C_VEL
LIN {X 0,Y 325.897,Z 742.076,A -85,B 0,C 180,E1 -25117.434,E2 -25117.434} C_VEL
LIN {X 0,Y 324.048,Z 741.057,A -85,B 0,C 180,E1 -25118.732,E2 -25118.732} C_VEL
LIN {X 0,Y 321.462,Z 739.579,A -85,B 0,C 180,E1 -25120.326,E2 -25120.326} C_VEL
LIN {X 0,Y 319.551,Z 738.329,A -85,B 0,C 180,E1 -25121.416,E2 -25121.416} C_VEL
LIN {X 0,Y 315.393,Z 735.363,A -85,B 0,C 180,E1 -25123.531,E2 -25123.531} C_VEL
LIN {X 0,Y 312.508,Z 733.492,A -85,B 0,C 180,E1 -25124.757,E2 -25124.757} C_VEL
LIN {X 0,Y 307.847,Z 730.628,A -85,B 0,C 180,E1 -25126.499,E2 -25126.499} C_VEL
LIN {X 0,Y 301.675,Z 726.306,A -85,B 0,C 180,E1 -25128.63,E2 -25128.63} C_VEL
LIN {X 0,Y 296.092,Z 722.365,A -85,B 0,C 180,E1 -25130.358,E2 -25130.358} C_VEL
LIN {X 0,Y 288.783,Z 717.257,A -85,B 0,C 180,E1 -25132.365,E2 -25132.365} C_VEL
LIN {X 0,Y 283.855,Z 713.608,A -85,B 0,C 180,E1 -25133.642,E2 -25133.642} C_VEL
LIN {X 0,Y 273.779,Z 706.252,A -85,B 0,C 180,E1 -25136.046,E2 -25136.046} C_VEL
LIN {X 0,Y 257.326,Z 694.23,A -85,B 0,C 180,E1 -25140.031,E2 -25140.031} C_VEL
LIN {X 0,Y 243.209,Z 682.67,A -85,B 0,C 180,E1 -25143.822,E2 -25143.822} C_VEL
LIN {X 0,Y 231.643,Z 671.206,A -85,B 0,C 180,E1 -25147.357,E2 -25147.357} C_VEL
LIN {X 0,Y 220.266,Z 658.013,A -85,B 0,C 180,E1 -25151.196,E2 -25151.196} C_VEL
LIN {X 0,Y 210.529,Z 644.761,A -85,B 0,C 180,E1 -25154.732,E2 -25154.732} C_VEL
LIN {X 0,Y 202.573,Z 632.249,A -85,B 0,C 180,E1 -25157.763,E2 -25157.763} C_VEL
LIN {X 0,Y 195.401,Z 618.387,A -85,B 0,C 180,E1 -25160.94,E2 -25160.94} C_VEL
LIN {X 0,Y 188.58,Z 602.319,A -85,B 0,C 180,E1 -25164.616,E2 -25164.616} C_VEL
LIN {X 0,Y 183.523,Z 591.926,A -85,B 0,C 180,E1 -25167.662,E2 -25167.662} C_VEL
LIN {X 0,Y 178.664,Z 583.134,A -85,B 0,C 180,E1 -25170.944,E2 -25170.944} C_VEL
LIN {X 0,Y 174.08,Z 575.709,A -85,B 0,C 180,E1 -25174.507,E2 -25174.507} C_VEL
LIN {X 0,Y 171.496,Z 571.77,A -85,B 0,C 180,E1 -25176.81,E2 -25176.81} C_VEL
LIN {X 0,Y 169.183,Z 568.289,A -85,B 0,C 180,E1 -25179.139,E2 -25179.139} C_VEL
LIN {X 0,Y 166.349,Z 564.156,A -85,B 0,C 180,E1 -25182.482,E2 -25182.482} C_VEL
LIN {X 0,Y 163.835,Z 560.647,A -85,B 0,C 180,E1 -25186.197,E2 -25186.197} C_VEL
LIN {X 0,Y 163.273,Z 559.525,A -85,B 0,C 180,E1 -25187.257,E2 -25187.257} C_VEL
LIN {X 0,Y 160.994,Z 557.042,A -85,B 0,C 180,E1 -25192.476,E2 -25192.476} C_VEL
LIN {X 0,Y 160.172,Z 554.751,A -85,B 0,C 180,E1 -25196.857,E2 -25196.857} C_VEL
LIN {X 0,Y 160.032,Z 554.174,A -85,B 0,C 180,E1 -25200.001,E2 -25200.001} C_VEL
LIN {X 0,Y 160.257,Z 554.986,A -85,B 0,C 180,E1 -25203.458,E2 -25203.458} C_VEL
LIN {X 0,Y 162.805,Z 559.194,A -85,B 0,C 180,E1 -25211.518,E2 -25211.518} C_VEL
LIN {X 0,Y 163.474,Z 559.869,A -85,B 0,C 180,E1 -25212.73,E2 -25212.73} C_VEL
LIN {X 0,Y 165.947,Z 563.729,A -85,B 0,C 180,E1 -25216.612,E2 -25216.612} C_VEL
LIN {X 0,Y 166.859,Z 564.912,A -85,B 0,C 180,E1 -25217.781,E2 -25217.781} C_VEL
LIN {X 0,Y 169.506,Z 568.63,A -85,B 0,C 180,E1 -25220.796,E2 -25220.796} C_VEL
LIN {X 0,Y 172.962,Z 573.976,A -85,B 0,C 180,E1 -25224.135,E2 -25224.135} C_VEL
LIN {X 0,Y 176.774,Z 579.998,A -85,B 0,C 180,E1 -25227.262,E2 -25227.262} C_VEL
LIN {X 0,Y 180.398,Z 587.991,A -85,B 0,C 180,E1 -25230.026,E2 -25230.026} C_VEL
LIN {X 0,Y 184.418,Z 598.057,A -85,B 0,C 180,E1 -25232.817,E2 -25232.817} C_VEL
LIN {X 0,Y 187.098,Z 605.716,A -85,B 0,C 180,E1 -25234.568,E2 -25234.568} C_VEL
LIN {X 0,Y 183.379,Z 650.724,A -85,B 0,C 180,E1 -25236.015,E2 -25236.015} C_VEL
LIN {X 0,Y 181.247,Z 664.319,A -85,B 0,C 180,E1 -25236.663,E2 -25236.663} C_VEL
LIN {X 0,Y 177.699,Z 679.3,A -85,B 0,C 180,E1 -25237.723,E2 -25237.723} C_VEL
LIN {X 0,Y 173.969,Z 691.413,A -85,B 0,C 180,E1 -25238.955,E2 -25238.955} C_VEL
LIN {X 0,Y 170.334,Z 701.328,A -85,B 0,C 180,E1 -25240.245,E2 -25240.245} C_VEL
LIN {X 0,Y 166.184,Z 711.046,A -85,B 0,C 180,E1 -25241.811,E2 -25241.811} C_VEL
LIN {X 0,Y 161.676,Z 720.46,A -85,B 0,C 180,E1 -25243.725,E2 -25243.725} C_VEL
LIN {X 0,Y 157.154,Z 729.079,A -85,B 0,C 180,E1 -25245.924,E2 -25245.924} C_VEL
LIN {X 0,Y 152.88,Z 736.453,A -85,B 0,C 180,E1 -25248.198,E2 -25248.198} C_VEL
LIN {X 0,Y 148.033,Z 743.969,A -85,B 0,C 180,E1 -25251.021,E2 -25251.021} C_VEL
LIN {X 0,Y 143.688,Z 750.442,A -85,B 0,C 180,E1 -25254.061,E2 -25254.061} C_VEL
LIN {X 0,Y 139.013,Z 756.981,A -85,B 0,C 180,E1 -25257.938,E2 -25257.938} C_VEL
LIN {X 0,Y 135.063,Z 762.417,A -85,B 0,C 180,E1 -25262.076,E2 -25262.076} C_VEL
LIN {X 0,Y 131.884,Z 766.868,A -85,B 0,C 180,E1 -25266.443,E2 -25266.443} C_VEL
LIN {X 0,Y 129.389,Z 770.42,A -85,B 0,C 180,E1 -25270.98,E2 -25270.98} C_VEL
LIN {X 0,Y 128.112,Z 772.366,A -85,B 0,C 180,E1 -25274.081,E2 -25274.081} C_VEL
LIN {X 0,Y 126.666,Z 775.068,A -85,B 0,C 180,E1 -25280.419,E2 -25280.419} C_VEL
LIN {X 0,Y 126.395,Z 775.895,A -85,B 0,C 180,E1 -25283.615,E2 -25283.615} C_VEL
LIN {X 0,Y 126.431,Z 776.635,A -85,B 0,C 180,E1 -25290,E2 -25290} C_VEL
LIN {X 0,Y 126.395,Z 775.895,A -85,B 0,C 180,E1 -25296.385,E2 -25296.385} C_VEL
LIN {X 0,Y 126.666,Z 775.068,A -85,B 0,C 180,E1 -25299.581,E2 -25299.581} C_VEL
LIN {X 0,Y 128.112,Z 772.366,A -85,B 0,C 180,E1 -25305.919,E2 -25305.919} C_VEL
LIN {X 0,Y 130.15,Z 769.402,A -85,B 0,C 180,E1 -25310.548,E2 -25310.548} C_VEL
LIN {X 0,Y 132.89,Z 765.569,A -85,B 0,C 180,E1 -25315.029,E2 -25315.029} C_VEL
LIN {X 0,Y 136.3,Z 760.8,A -85,B 0,C 180,E1 -25319.33,E2 -25319.33} C_VEL
LIN {X 0,Y 141.256,Z 753.854,A -85,B 0,C 180,E1 -25324.036,E2 -25324.036} C_VEL
LIN {X 0,Y 146.205,Z 746.643,A -85,B 0,C 180,E1 -25327.797,E2 -25327.797} C_VEL
LIN {X 0,Y 150.91,Z 739.574,A -85,B 0,C 180,E1 -25330.691,E2 -25330.691} C_VEL
LIN {X 0,Y 155.799,Z 731.507,A -85,B 0,C 180,E1 -25333.363,E2 -25333.363} C_VEL
LIN {X 0,Y 160.021,Z 723.855,A -85,B 0,C 180,E1 -25335.444,E2 -25335.444} C_VEL
LIN {X 0,Y 164.511,Z 714.766,A -85,B 0,C 180,E1 -25337.469,E2 -25337.469} C_VEL
LIN {X 0,Y 168.556,Z 705.719,A -85,B 0,C 180,E1 -25339.087,E2 -25339.087} C_VEL
LIN {X 0,Y 171.002,Z 699.582,A -85,B 0,C 180,E1 -25340.033,E2 -25340.033} C_VEL
LIN {X 0,Y 172.544,Z 694.484,A -85,B 0,C 180,E1 -25340.89,E2 -25340.89} C_VEL
LIN {X 0,Y 173.605,Z 686.026,A -85,B 0,C 180,E1 -25342.572,E2 -25342.572} C_VEL
LIN {X 0,Y 174.308,Z 678.187,A -85,B 0,C 180,E1 -25343.958,E2 -25343.958} C_VEL
LIN {X 0,Y 175.373,Z 671.753,A -85,B 0,C 180,E1 -25344.683,E2 -25344.683} C_VEL
LIN {X 0,Y 177.582,Z 661.385,A -85,B 0,C 180,E1 -25345.328,E2 -25345.328} C_VEL
LIN {X 0,Y 179.254,Z 650.7,A -85,B 0,C 180,E1 -25345.809,E2 -25345.809} C_VEL
LIN {X 0,Y 182.12,Z 618.836,A -85,B 0,C 180,E1 -25346.824,E2 -25346.824} C_VEL
LIN {X 0,Y 182.92,Z 608.169,A -85,B 0,C 180,E1 -25347.191,E2 -25347.191} C_VEL
LIN {X 0,Y 179.168,Z 597.478,A -85,B 0,C 180,E1 -25349.909,E2 -25349.909} C_VEL
LIN {X 0,Y 175.428,Z 588.316,A -85,B 0,C 180,E1 -25352.861,E2 -25352.861} C_VEL
LIN {X 0,Y 173.631,Z 584.693,A -85,B 0,C 180,E1 -25354.367,E2 -25354.367} C_VEL
LIN {X 0,Y 169.704,Z 578.218,A -85,B 0,C 180,E1 -25357.956,E2 -25357.956} C_VEL
LIN {X 0,Y 167.426,Z 574.717,A -85,B 0,C 180,E1 -25360.377,E2 -25360.377} C_VEL
LIN {X 0,Y 164.644,Z 570.542,A -85,B 0,C 180,E1 -25363.89,E2 -25363.89} C_VEL
LIN {X 0,Y 162.263,Z 566.762,A -85,B 0,C 180,E1 -25367.809,E2 -25367.809} C_VEL
LIN {X 0,Y 159.233,Z 561.535,A -85,B 0,C 180,E1 -25378.102,E2 -25378.102} C_VEL
LIN {X 0,Y 159.171,Z 561.182,A -85,B 0,C 180,E1 -25379.999,E2 -25379.999} C_VEL
LIN {X 0,Y 159.367,Z 562.137,A -85,B 0,C 180,E1 -25383.792,E2 -25383.792} C_VEL
LIN {X 0,Y 161.561,Z 566.067,A -85,B 0,C 180,E1 -25391.237,E2 -25391.237} C_VEL
LIN {X 0,Y 162.303,Z 566.828,A -85,B 0,C 180,E1 -25392.662,E2 -25392.662} C_VEL
LIN {X 0,Y 164.641,Z 570.591,A -85,B 0,C 180,E1 -25396.506,E2 -25396.506} C_VEL
LIN {X 0,Y 165.679,Z 572.151,A -85,B 0,C 180,E1 -25397.91,E2 -25397.91} C_VEL
LIN {X 0,Y 168.387,Z 576.187,A -85,B 0,C 180,E1 -25401.077,E2 -25401.077} C_VEL
LIN {X 0,Y 171.075,Z 580.515,A -85,B 0,C 180,E1 -25403.771,E2 -25403.771} C_VEL
LIN {X 0,Y 174.706,Z 586.488,A -85,B 0,C 180,E1 -25406.907,E2 -25406.907} C_VEL
LIN {X 0,Y 179.247,Z 594.712,A -85,B 0,C 180,E1 -25410.311,E2 -25410.311} C_VEL
LIN {X 0,Y 183.574,Z 603.677,A -85,B 0,C 180,E1 -25413.199,E2 -25413.199} C_VEL
LIN {X 0,Y 187.516,Z 612.92,A -85,B 0,C 180,E1 -25415.613,E2 -25415.613} C_VEL
LIN {X 0,Y 194.412,Z 628.988,A -85,B 0,C 180,E1 -25419.309,E2 -25419.309} C_VEL
LIN {X 0,Y 202.027,Z 642.915,A -85,B 0,C 180,E1 -25422.706,E2 -25422.706} C_VEL
LIN {X 0,Y 208.991,Z 653.758,A -85,B 0,C 180,E1 -25425.595,E2 -25425.595} C_VEL
LIN {X 0,Y 217.123,Z 664.882,A -85,B 0,C 180,E1 -25428.812,E2 -25428.812} C_VEL
LIN {X 0,Y 227.666,Z 677.241,A -85,B 0,C 180,E1 -25432.644,E2 -25432.644} C_VEL
LIN {X 0,Y 239.903,Z 689.205,A -85,B 0,C 180,E1 -25436.605,E2 -25436.605} C_VEL
LIN {X 0,Y 254.121,Z 700.533,A -85,B 0,C 180,E1 -25440.593,E2 -25440.593} C_VEL
LIN {X 0,Y 268.945,Z 711.227,A -85,B 0,C 180,E1 -25444.36,E2 -25444.36} C_VEL
LIN {X 0,Y 279.039,Z 718.333,A -85,B 0,C 180,E1 -25446.823,E2 -25446.823} C_VEL
LIN {X 0,Y 286.444,Z 723.756,A -85,B 0,C 180,E1 -25448.8,E2 -25448.8} C_VEL
LIN {X 0,Y 291.775,Z 727.428,A -85,B 0,C 180,E1 -25450.293,E2 -25450.293} C_VEL
LIN {X 0,Y 297.505,Z 731.488,A -85,B 0,C 180,E1 -25452.116,E2 -25452.116} C_VEL
LIN {X 0,Y 302.421,Z 734.873,A -85,B 0,C 180,E1 -25453.808,E2 -25453.808} C_VEL
LIN {X 0,Y 308.554,Z 738.694,A -85,B 0,C 180,E1 -25456.163,E2 -25456.163} C_VEL
LIN {X 0,Y 310.242,Z 739.856,A -85,B 0,C 180,E1 -25456.925,E2 -25456.925} C_VEL
LIN {X 0,Y 314.722,Z 742.98,A -85,B 0,C 180,E1 -25459.278,E2 -25459.278} C_VEL
LIN {X 0,Y 317.769,Z 744.837,A -85,B 0,C 180,E1 -25461.094,E2 -25461.094} C_VEL
LIN {X 0,Y 319.738,Z 745.893,A -85,B 0,C 180,E1 -25462.422,E2 -25462.422} C_VEL
LIN {X 0,Y 321.417,Z 746.74,A -85,B 0,C 180,E1 -25463.724,E2 -25463.724} C_VEL
LIN {X 0,Y 322.751,Z 747.386,A -85,B 0,C 180,E1 -25465.003,E2 -25465.003} C_VEL
LIN {X 0,Y 323.942,Z 747.814,A -85,B 0,C 180,E1 -25466.346,E2 -25466.346} C_VEL
LIN {X 0,Y 324.661,Z 748.106,A -85,B 0,C 180,E1 -25467.519,E2 -25467.519} C_VEL
LIN {X 0,Y 325.128,Z 748.292,A -85,B 0,C 180,E1 -25468.761,E2 -25468.761} C_VEL
LIN {X 0,Y 325.375,Z 748.296,A -85,B 0,C 180,E1 -25470,E2 -25470} C_VEL
LIN {X 0,Y 325.125,Z 748.294,A -85,B 0,C 180,E1 -25471.239,E2 -25471.239} C_VEL
LIN {X 0,Y 324.662,Z 748.11,A -85,B 0,C 180,E1 -25472.481,E2 -25472.481} C_VEL
LIN {X 0,Y 323.866,Z 747.811,A -85,B 0,C 180,E1 -25473.733,E2 -25473.733} C_VEL
LIN {X 0,Y 322.775,Z 747.367,A -85,B 0,C 180,E1 -25474.996,E2 -25474.996} C_VEL
LIN {X 0,Y 321.41,Z 746.73,A -85,B 0,C 180,E1 -25476.277,E2 -25476.277} C_VEL
LIN {X 0,Y 319.275,Z 745.671,A -85,B 0,C 180,E1 -25477.886,E2 -25477.886} C_VEL
LIN {X 0,Y 315.546,Z 743.513,A -85,B 0,C 180,E1 -25480.264,E2 -25480.264} C_VEL
LIN {X 0,Y 313.024,Z 741.818,A -85,B 0,C 180,E1 -25481.658,E2 -25481.658} C_VEL
LIN {X 0,Y 308.57,Z 738.696,A -85,B 0,C 180,E1 -25483.836,E2 -25483.836} C_VEL
LIN {X 0,Y 304.645,Z 736.275,A -85,B 0,C 180,E1 -25485.384,E2 -25485.384} C_VEL
LIN {X 0,Y 297.589,Z 731.558,A -85,B 0,C 180,E1 -25487.879,E2 -25487.879} C_VEL
LIN {X 0,Y 291.394,Z 727.163,A -85,B 0,C 180,E1 -25489.846,E2 -25489.846} C_VEL
LIN {X 0,Y 283.435,Z 721.605,A -85,B 0,C 180,E1 -25492.025,E2 -25492.025} C_VEL
LIN {X 0,Y 276.488,Z 716.595,A -85,B 0,C 180,E1 -25493.786,E2 -25493.786} C_VEL
LIN {X 0,Y 266.464,Z 709.417,A -85,B 0,C 180,E1 -25496.268,E2 -25496.268} C_VEL
LIN {X 0,Y 250.784,Z 698.084,A -85,B 0,C 180,E1 -25500.293,E2 -25500.293} C_VEL
LIN {X 0,Y 236.891,Z 686.497,A -85,B 0,C 180,E1 -25504.31,E2 -25504.31} C_VEL
LIN {X 0,Y 226.589,Z 676.021,A -85,B 0,C 180,E1 -25507.73,E2 -25507.73} C_VEL
LIN {X 0,Y 217.123,Z 664.885,A -85,B 0,C 180,E1 -25511.188,E2 -25511.188} C_VEL
LIN {X 0,Y 208.265,Z 652.683,A -85,B 0,C 180,E1 -25514.704,E2 -25514.704} C_VEL
LIN {X 0,Y 200.625,Z 640.535,A -85,B 0,C 180,E1 -25517.914,E2 -25517.914} C_VEL
LIN {X 0,Y 192.905,Z 625.818,A -85,B 0,C 180,E1 -25521.43,E2 -25521.43} C_VEL
LIN {X 0,Y 184.96,Z 606.694,A -85,B 0,C 180,E1 -25525.939,E2 -25525.939} C_VEL
LIN {X 0,Y 180.467,Z 597.105,A -85,B 0,C 180,E1 -25528.847,E2 -25528.847} C_VEL
LIN {X 0,Y 175.928,Z 588.631,A -85,B 0,C 180,E1 -25532.128,E2 -25532.128} C_VEL
LIN {X 0,Y 171.791,Z 581.624,A -85,B 0,C 180,E1 -25535.577,E2 -25535.577} C_VEL
LIN {X 0,Y 169.14,Z 577.441,A -85,B 0,C 180,E1 -25538.123,E2 -25538.123} C_VEL
LIN {X 0,Y 167.334,Z 574.617,A -85,B 0,C 180,E1 -25540.084,E2 -25540.084} C_VEL
LIN {X 0,Y 164.808,Z 570.755,A -85,B 0,C 180,E1 -25543.272,E2 -25543.272} C_VEL
LIN {X 0,Y 162.377,Z 567.01,A -85,B 0,C 180,E1 -25547.185,E2 -25547.185} C_VEL
LIN {X 0,Y 161.997,Z 566.379,A -85,B 0,C 180,E1 -25547.933,E2 -25547.933} C_VEL
LIN {X 0,Y 159.595,Z 563.018,A -85,B 0,C 180,E1 -25554.632,E2 -25554.632} C_VEL
LIN {X 0,Y 159.244,Z 561.653,A -85,B 0,C 180,E1 -25557.472,E2 -25557.472} C_VEL
LIN {X 0,Y 159.166,Z 561.229,A -85,B 0,C 180,E1 -25560.001,E2 -25560.001} C_VEL
LIN {X 0,Y 159.379,Z 562.147,A -85,B 0,C 180,E1 -25563.477,E2 -25563.477} C_VEL
LIN {X 0,Y 161.787,Z 566.186,A -85,B 0,C 180,E1 -25571.274,E2 -25571.274} C_VEL
LIN {X 0,Y 162.336,Z 566.941,A -85,B 0,C 180,E1 -25572.344,E2 -25572.344} C_VEL
LIN {X 0,Y 164.864,Z 570.782,A -85,B 0,C 180,E1 -25576.406,E2 -25576.406} C_VEL
LIN {X 0,Y 168.535,Z 576.405,A -85,B 0,C 180,E1 -25580.841,E2 -25580.841} C_VEL
LIN {X 0,Y 171.224,Z 580.7,A -85,B 0,C 180,E1 -25583.511,E2 -25583.511} C_VEL
LIN {X 0,Y 174.526,Z 586.23,A -85,B 0,C 180,E1 -25586.373,E2 -25586.373} C_VEL
LIN {X 0,Y 178.548,Z 595.882,A -85,B 0,C 180,E1 -25589.622,E2 -25589.622} C_VEL
LIN {X 0,Y 182.174,Z 605.884,A -85,B 0,C 180,E1 -25592.282,E2 -25592.282} C_VEL
LIN {X 0,Y 182.92,Z 608.143,A -85,B 0,C 180,E1 -25592.807,E2 -25592.807} C_VEL
LIN {X 0,Y 179.36,Z 649.879,A -85,B 0,C 180,E1 -25594.146,E2 -25594.146} C_VEL
LIN {X 0,Y 177.427,Z 662.298,A -85,B 0,C 180,E1 -25594.724,E2 -25594.724} C_VEL
LIN {X 0,Y 174.484,Z 675.541,A -85,B 0,C 180,E1 -25595.599,E2 -25595.599} C_VEL
LIN {X 0,Y 170.208,Z 689.461,A -85,B 0,C 180,E1 -25596.871,E2 -25596.871} C_VEL
LIN {X 0,Y 165.821,Z 701.129,A -85,B 0,C 180,E1 -25598.365,E2 -25598.365} C_VEL
LIN {X 0,Y 161.536,Z 710.848,A -85,B 0,C 180,E1 -25599.933,E2 -25599.933} C_VEL
LIN {X 0,Y 156.828,Z 720.261,A -85,B 0,C 180,E1 -25601.841,E2 -25601.841} C_VEL
LIN {X 0,Y 152.286,Z 728.566,A -85,B 0,C 180,E1 -25603.959,E2 -25603.959} C_VEL
LIN {X 0,Y 147.628,Z 736.253,A -85,B 0,C 180,E1 -25606.348,E2 -25606.348} C_VEL
LIN {X 0,Y 142.573,Z 743.771,A -85,B 0,C 180,E1 -25609.222,E2 -25609.222} C_VEL
LIN {X 0,Y 137.946,Z 750.242,A -85,B 0,C 180,E1 -25612.313,E2 -25612.313} C_VEL
LIN {X 0,Y 133.017,Z 756.782,A -85,B 0,C 180,E1 -25616.306,E2 -25616.306} C_VEL
LIN {X 0,Y 128.794,Z 762.218,A -85,B 0,C 180,E1 -25620.587,E2 -25620.587} C_VEL
LIN {X 0,Y 125.364,Z 766.669,A -85,B 0,C 180,E1 -25625.137,E2 -25625.137} C_VEL
LIN {X 0,Y 122.67,Z 770.221,A -85,B 0,C 180,E1 -25629.895,E2 -25629.895} C_VEL
LIN {X 0,Y 121.249,Z 772.166,A -85,B 0,C 180,E1 -25633.153,E2 -25633.153} C_VEL
LIN {X 0,Y 119.644,Z 774.869,A -85,B 0,C 180,E1 -25639.85,E2 -25639.85} C_VEL
LIN {X 0,Y 119.223,Z 776.178,A -85,B 0,C 180,E1 -25646.621,E2 -25646.621} C_VEL
LIN {X 0,Y 119.336,Z 776.437,A -85,B 0,C 180,E1 -25650,E2 -25650} C_VEL
LIN {X 0,Y 119.307,Z 775.696,A -85,B 0,C 180,E1 -25656.766,E2 -25656.766} C_VEL
LIN {X 0,Y 119.644,Z 774.869,A -85,B 0,C 180,E1 -25660.15,E2 -25660.15} C_VEL
LIN {X 0,Y 121.248,Z 772.166,A -85,B 0,C 180,E1 -25666.847,E2 -25666.847} C_VEL
LIN {X 0,Y 123.477,Z 769.203,A -85,B 0,C 180,E1 -25671.713,E2 -25671.713} C_VEL
LIN {X 0,Y 126.422,Z 765.369,A -85,B 0,C 180,E1 -25676.405,E2 -25676.405} C_VEL
LIN {X 0,Y 130.119,Z 760.601,A -85,B 0,C 180,E1 -25680.871,E2 -25680.871} C_VEL
LIN {X 0,Y 135.404,Z 753.655,A -85,B 0,C 180,E1 -25685.726,E2 -25685.726} C_VEL
LIN {X 0,Y 139.707,Z 747.78,A -85,B 0,C 180,E1 -25688.962,E2 -25688.962} C_VEL
LIN {X 0,Y 145.58,Z 739.376,A -85,B 0,C 180,E1 -25692.52,E2 -25692.52} C_VEL
LIN {X 0,Y 150.602,Z 731.48,A -85,B 0,C 180,E1 -25695.17,E2 -25695.17} C_VEL
LIN {X 0,Y 155.196,Z 723.442,A -85,B 0,C 180,E1 -25697.38,E2 -25697.38} C_VEL
LIN {X 0,Y 159.776,Z 714.567,A -85,B 0,C 180,E1 -25699.354,E2 -25699.354} C_VEL
LIN {X 0,Y 163.987,Z 705.521,A -85,B 0,C 180,E1 -25700.965,E2 -25700.965} C_VEL
LIN {X 0,Y 168.302,Z 694.72,A -85,B 0,C 180,E1 -25702.503,E2 -25702.503} C_VEL
LIN {X 0,Y 171.856,Z 684.469,A -85,B 0,C 180,E1 -25703.62,E2 -25703.62} C_VEL
LIN {X 0,Y 174.777,Z 674.18,A -85,B 0,C 180,E1 -25704.514,E2 -25704.514} C_VEL
LIN {X 0,Y 175.373,Z 671.753,A -85,B 0,C 180,E1 -25704.683,E2 -25704.683} C_VEL
LIN {X 0,Y 176.369,Z 666.154,A -85,B 0,C 180,E1 -25705.231,E2 -25705.231} C_VEL
LIN {X 0,Y 176.382,Z 657.028,A -85,B 0,C 180,E1 -25706.495,E2 -25706.495} C_VEL
LIN {X 0,Y 176.096,Z 647.774,A -85,B 0,C 180,E1 -25707.654,E2 -25707.654} C_VEL
LIN {X 0,Y 176.331,Z 641.978,A -85,B 0,C 180,E1 -25708.02,E2 -25708.02} C_VEL
LIN {X 0,Y 178.925,Z 610.754,A -85,B 0,C 180,E1 -25709.02,E2 -25709.02} C_VEL
LIN {X 0,Y 175.798,Z 601.493,A -85,B 0,C 180,E1 -25711.51,E2 -25711.51} C_VEL
LIN {X 0,Y 172.03,Z 591.827,A -85,B 0,C 180,E1 -25714.802,E2 -25714.802} C_VEL
LIN {X 0,Y 167.978,Z 584.744,A -85,B 0,C 180,E1 -25718.685,E2 -25718.685} C_VEL
LIN {X 0,Y 165.541,Z 580.956,A -85,B 0,C 180,E1 -25721.432,E2 -25721.432} C_VEL
LIN {X 0,Y 163.245,Z 577.263,A -85,B 0,C 180,E1 -25724.55,E2 -25724.55} C_VEL
LIN {X 0,Y 160.771,Z 573.19,A -85,B 0,C 180,E1 -25728.973,E2 -25728.973} C_VEL
LIN {X 0,Y 158.365,Z 568.616,A -85,B 0,C 180,E1 -25738.091,E2 -25738.091} C_VEL
LIN {X 0,Y 158.296,Z 568.339,A -85,B 0,C 180,E1 -25740.635,E2 -25740.635} C_VEL
LIN {X 0,Y 158.457,Z 569.133,A -85,B 0,C 180,E1 -25743.495,E2 -25743.495} C_VEL
LIN {X 0,Y 160.416,Z 572.952,A -85,B 0,C 180,E1 -25750.704,E2 -25750.704} C_VEL
LIN {X 0,Y 161.066,Z 573.6,A -85,B 0,C 180,E1 -25752.025,E2 -25752.025} C_VEL
LIN {X 0,Y 163.297,Z 577.359,A -85,B 0,C 180,E1 -25755.923,E2 -25755.923} C_VEL
LIN {X 0,Y 166.639,Z 582.612,A -85,B 0,C 180,E1 -25760.246,E2 -25760.246} C_VEL
LIN {X 0,Y 170.329,Z 588.734,A -85,B 0,C 180,E1 -25764.044,E2 -25764.044} C_VEL
LIN {X 0,Y 175.056,Z 597.421,A -85,B 0,C 180,E1 -25768.088,E2 -25768.088} C_VEL
LIN {X 0,Y 179.465,Z 606.534,A -85,B 0,C 180,E1 -25771.338,E2 -25771.338} C_VEL
LIN {X 0,Y 183.599,Z 616.495,A -85,B 0,C 180,E1 -25774.102,E2 -25774.102} C_VEL
LIN {X 0,Y 190.455,Z 633.243,A -85,B 0,C 180,E1 -25778.078,E2 -25778.078} C_VEL
LIN {X 0,Y 198.312,Z 648.317,A -85,B 0,C 180,E1 -25781.909,E2 -25781.909} C_VEL
LIN {X 0,Y 206.043,Z 660.829,A -85,B 0,C 180,E1 -25785.506,E2 -25785.506} C_VEL
LIN {X 0,Y 214.15,Z 672.031,A -85,B 0,C 180,E1 -25789.008,E2 -25789.008} C_VEL
LIN {X 0,Y 224.362,Z 684.053,A -85,B 0,C 180,E1 -25793.011,E2 -25793.011} C_VEL
LIN {X 0,Y 235.292,Z 694.582,A -85,B 0,C 180,E1 -25796.754,E2 -25796.754} C_VEL
